(* IEC 61131-3 sources: Mizera_Tube/Plc (part 11) *)

(* ---- DataInterp.plc ---- *)
*******************************************************************************
*   DataInterp.plc
*   ESAutomotion
*   LASER machine
*******************************************************************************
#funcdec "DynMng.plc"

VAR
#include "Cnc.inc"

END_VAR

VAR_IN_OUT
#include "mem.inc"
END_VAR

#include "Iol.inc"

VAR_IN_OUT
A_CUT_DISTANCE          AT %L_CutDistance;
A_CUT_PRESSURE          AT %L_CutPressure;
A_CUT_FOCAL             AT %L_CutFocal;
A_CUT_FEED              AT %L_FeedA;
A_CUT_POWER             AT %L_CutPower;
A_CUT_DUTY              AT %L_CutDuty;
A_OPTION_FUN_SPEED      AT %L_SourceInt16;
A_OPTION_ENAB           AT %L_SourceInt16;
END_VAR

VAR
END_VAR

*******************************************************************************
*   Calcola dati di taglio tramite interpolazione lineare tra 2 linee di taglio
*
*       Formula: Y = Y1 + ( ((X-X1)/(X2-X1)) * (Y2-Y1) )
*******************************************************************************
FUNCTION_BLOCK LSR_DATA_INTERP

VAR_INPUT
xAngle:         DWORD;      * degree x 1000
xCutLineInd:    DWORD;      *
xFir:           DWORD;      *
END_VAR

VAR_OUTPUT
yCutPower:      DWORD;
yCutDuty:       DWORD;
yCutPressure:   DWORD;
yCutFocal:      DWORD;
yCutDistance:   DWORD;
yCutFeed:       DWORD;
yCutFeedPerc:   DWORD;
yFirstLine:     DWORD;
ySecondLine:    DWORD;
END_VAR

VAR
lAngleABS:      DWORD;
lFirstCutLine:  DWORD;
lSecondCutLine: DWORD;
l_x1:           DWORD;
l_x2:           DWORD;
l_y1:           DWORD;
l_y2:           DWORD;
l_x_x1:         DWORD;
l_x2_x1:        DWORD;
l_y2_y1:        DWORD;
POWER_CALC:     POINTS_INT_CALC;
POWER_CALC2:    POINTS_INT_CALC;
DUTY_CALC:      POINTS_INT_CALC;
DUTY_CALC2:     POINTS_INT_CALC;
Fir1:           DWORD;
flgerror_fir1:  DWORD;
RTRIG_FIR_INIT: R_TRIG;
l_CutFeedPerc:  DWORD;
ltemp:          DWORD;
END_VAR
***************************************

CAL  RTRIG_FIR_INIT (CLK:=%cn0.rc8.0)
LD   RTRIG_FIR_INIT.Q
JMPCN no_init_fir

LD   xFir
DIV  %plc0.PlcCycle
ST   Fir1
LD   0
FIR_INIT (INS=7, LEN=Fir1)
ST   flgerror_fir1             * 0 = OK

no_init_fir:
LD   xAngle
ABS
ST   lAngleABS

LD   lAngleABS
GE   30000
JMPCN no_30
LD   5
ST   lFirstCutLine
LD   6
ST   lSecondCutLine

LD   30000
ST   l_x1
LD   45000
ST   l_x2
JMP  com_a

no_30:
LD   lAngleABS
GE   15000
JMPCN no_15
LD   xCutLineInd
ST   lFirstCutLine
LD   5
ST   lSecondCutLine
LD   15000
ST   l_x1
LD   30000
ST   l_x2
JMP  com_a

no_15:
LD   xCutLineInd
ST   lFirstCutLine
ST   lSecondCutLine
LD   0
ST   l_x1
LD   15000
ST   l_x2

com_a:
LD   lAngleABS
SUB  l_x1
ST   l_x_x1
LD   l_x2
SUB  l_x1
ST   l_x2_x1

LD   lFirstCutLine
ST   yFirstLine
LD   lSecondCutLine
ST   ySecondLine

***************************************
*   Pressione
***************************************
PATH %TabLsr[lFirstCutLine]
LD   A_CUT_PRESSURE
ST   l_y1

PATH %TabLsr[lSecondCutLine]
LD   A_CUT_PRESSURE
ST   l_y2

LD   l_y2
SUB  l_y1
ST   l_y2_y1

LD   l_x_x1
MULDIV(M=l_y2_y1,D=l_x2_x1)
ADD  l_y1
ST   yCutPressure

***************************************
*   Focale
***************************************
PATH %TabLsr[lFirstCutLine]
LD   A_CUT_FOCAL
ST   l_y1

PATH %TabLsr[lSecondCutLine]
LD   A_CUT_FOCAL
ST   l_y2

LD   l_y2
SUB  l_y1
ST   l_y2_y1

LD   l_x_x1
MULDIV(M=l_y2_y1,D=l_x2_x1)
ADD  l_y1
ST   yCutFocal

***************************************
*   Altezza di taglio
***************************************
PATH %TabLsr[lFirstCutLine]
LD   A_CUT_DISTANCE
ST   l_y1

PATH %TabLsr[lSecondCutLine]
LD   A_CUT_DISTANCE
ST   l_y2

LD   l_y2
SUB  l_y1
ST   l_y2_y1

LD   l_x_x1
MULDIV(M=l_y2_y1,D=l_x2_x1)
ADD  l_y1
ST   yCutDistance

***************************************
*   Velocita' di taglio
*   - yCutFeed  [mm/min]
*   - yCutFeedPerc  [%] rispetto a linea taglio no bevel
***************************************
***todo PATH %TabLsr[lFirstCutLine]
PATH %TabLsr[1]
LD   A_CUT_FEED
ST   l_y1

PATH %TabLsr[lSecondCutLine]
LD   A_CUT_FEED
ST   l_y2

LD   l_y2
SUB  l_y1
ST   l_y2_y1

LD   lAngleABS
ST   l_x_x1
LD   l_x2
ST   l_x2_x1

LD   l_x_x1
MULDIV(M=l_y2_y1,D=l_x2_x1)
ADD  l_y1
ST   yCutFeed

LD   100            * 100%
ST   l_CutFeedPerc

LD   yCutFeed
MUL  100
DIV  l_y1
ST   l_CutFeedPerc

***todo
***LD   l_y2_y1
***EQ   0
***JMPC f_eq
***LD   yCutFeed
***SUB  l_y1
***MUL  100
***DIV  l_y2_y1

LD   0                       * N/C
FIR_RUN (INS=7, X=l_CutFeedPerc)
ST   ltemp

LD   l_CutFeedPerc
EQ   2147483647
JMPCN no_err_1

LD   ltemp
ST   l_CutFeedPerc

no_err_1:
f_eq:
LD   l_CutFeedPerc
ST   yCutFeedPerc

***************************************
*   Potenza
***************************************
PATH %TabLsr[lFirstCutLine]

LD   A_CUT_POWER
ST   l_y1

LD   A_OPTION_FUN_SPEED.3
JMPCN no_pow_funspeed

LD   PercInterpSpeed
ST   POWER_CALC.xPercSpeed
LD   lFirstCutLine
ST   POWER_CALC.xCutLineInd
LD   1
ST   POWER_CALC.xCodTec             * Tecnology 0=duty 1=power 2=frequency

CAL  POWER_CALC

LD   POWER_CALC.yResult
DIV  1000
MUL  A_CUT_POWER
DIV  100
ST   l_y1

no_pow_funspeed:

PATH %TabLsr[lSecondCutLine]
LD   A_CUT_POWER
ST   l_y2

LD   A_OPTION_FUN_SPEED.3           * enab power=funz(speed)
JMPCN no_pow_funspeed2

LD   PercInterpSpeed
ST   POWER_CALC2.xPercSpeed
LD   lSecondCutLine
ST   POWER_CALC2.xCutLineInd
LD   1
ST   POWER_CALC2.xCodTec            * 0=duty 1=power 2=frequency

CAL  POWER_CALC2

LD   POWER_CALC2.yResult
DIV  1000
MUL  A_CUT_POWER
DIV  100
ST   l_y2

no_pow_funspeed2:
LD   l_y2
SUB  l_y1
ST   l_y2_y1

LD   l_x_x1
MULDIV(M=l_y2_y1,D=l_x2_x1)
ADD  l_y1
ST   yCutPower

***************************************
*   Duty
***************************************
PATH %TabLsr[lFirstCutLine]

LD   A_CUT_DUTY
ST   l_y1

LD   A_OPTION_FUN_SPEED.2           * enab duty=funz(speed)
JMPCN no_duty_funspeed

LD   PercInterpSpeed
ST   DUTY_CALC.xPercSpeed
LD   lFirstCutLine
ST   DUTY_CALC.xCutLineInd
LD   0
ST   DUTY_CALC.xCodTec              * 0=duty 1=power 2=frequency

CAL  DUTY_CALC

LD   DUTY_CALC.yResult
DIV  1000
MUL  A_CUT_DUTY
DIV  100
ST   l_y1

no_duty_funspeed:
PATH %TabLsr[lSecondCutLine]
LD   A_CUT_DUTY
ST   l_y2

LD   A_OPTION_FUN_SPEED.2           * enab duty=funz(speed)
JMPCN no_duty_funspeed2

LD   PercInterpSpeed
ST   DUTY_CALC2.xPercSpeed
LD   lSecondCutLine
ST   DUTY_CALC2.xCutLineInd
LD   0
ST   DUTY_CALC2.xCodTec             * 0=duty 1=power 2=frequency

CAL  DUTY_CALC2

LD   DUTY_CALC2.yResult
DIV  1000
MUL  A_CUT_DUTY
DIV  100
ST   l_y2

no_duty_funspeed2:
LD   l_y2
SUB  l_y1
ST   l_y2_y1

LD   l_x_x1
MULDIV(M=l_y2_y1,D=l_x2_x1)
ADD  l_y1
ST   yCutDuty

END_FUNCTION_BLOCK

*******************************************************************************
*   Calcola dati di taglio in base all'angolo utilizzando le pd_spline
*   dedicate nell'attuale linea di taglio selezionata
*
*NB:
*pd_spline[150]     potenza linea 1    	(L_SourceInt16.8=abilitazione)
*pd_spline[151]		velocità linea 1	(L_SourceInt16.9=abilitazione)
*pd_spline[152]		altezza linea 1	    (L_SourceInt16.10=abilitazione)
*pd_spline[153]		focale linea 1	    (L_SourceInt16.11=abilitazione)
*pd_spline[154]		duty linea 1	    (L_SourceInt16.12=abilitazione)
*pd_spline[155]		gas linea 1		    (L_SourceInt16.13=abilitazione)
*pd_spline[156]		... linea 1         (L_SourceInt16.14=abilitazione)
*
* NB: Usa variabili globali SOLO per la simulazione (PER TEST USO INTERNO!)
* NB: %LSRPlcOp0.3 -> Enab function
*******************************************************************************
FUNCTION_BLOCK LSRDATACALC_ANGLE

VAR_INPUT
xAngle:         DWORD;      * degree x 1000
xCutLineInd:    DWORD;      * cutting line selected (1-10)
END_VAR

VAR_OUTPUT
yCutPower:      DWORD;      * % x 1000
yCutDuty:       DWORD;      * % x 1000
yCutFocal:      DWORD;      * % x 1000
yCutCuth:       DWORD;      * % x 1000
yCutGas:        DWORD;      * % x 1000
END_VAR

VAR
lAngleABS:      DWORD;
pdspline_num:   DWORD;
tmpPower:       DWORD;
tmpDuty:        DWORD;
tmpFocal:       DWORD;
tmpCuth:        DWORD;
tmpGas:         DWORD;
ANGLE_POWER_CALC:   LINEAR_CALC;
ANGLE_DUTY_CALC:    LINEAR_CALC;
ANGLE_FOCAL_CALC:   LINEAR_CALC;
ANGLE_CUTH_CALC:    LINEAR_CALC;
ANGLE_GAS_CALC:     LINEAR_CALC;
END_VAR
***************************************

*** SOLO per SIMULAZIONE INTERNA
LD   %TsCutDataLinear.CDL_SimOnPsw
EQ   2021
JMPCN no_sim_datainterp

LD   %TsCutDataLinear.CDL_SimAngle
ST   lAngleABS

LD   1
ST   xCutLineInd            * 1 per solo TEST !

JMP  initf

no_sim_datainterp:
LD   xAngle
ABS
ST   lAngleABS

initf:
PATH %TabLsr[xCutLineInd]

* Cuttting lines 1,2,3
LD   xCutLineInd
SUB  1
MUL  7                      * numero pd_spline[] per ciascuna linea di taglio
ADD  150
ST   pdspline_num           * 150 pd_spline linea1, 157 pd_spline linea2.....

* Cutting lines 11,12,13
LD   xCutLineInd
GT   10
JMPCN FROM11TO15
     LD   xCutLineInd
     SUB  11
     MUL  7                 * numero pd_spline[] per ciascuna linea di taglio
     ADD  180
     ST   pdspline_num      * 180 pd_spline linea1, 157 pd_spline linea2.....
FROM11TO15:

***************************************
*   POTENZA
*   pd_spline[150]=linea 1
*   Il valore trovato è l'incremento o
*   decremento della potenza attuale
***************************************
LD   0
ST   tmpPower

LD   A_OPTION_ENAB.8
AND  %LSRPlcOp0.3                       * Enab data cutting interpolation
AND  IncaseofbevelCut
JMPCN dato_ko

LD   lAngleABS
ST   ANGLE_POWER_CALC.xInput

LD   pdspline_num
ST   ANGLE_POWER_CALC.xIndex

CAL  ANGLE_POWER_CALC

LD   ANGLE_POWER_CALC.yResult
EQ   2147483647
JMPC dato_ko

LD   ANGLE_POWER_CALC.yResult
ST   tmpPower

dato_ko:
LD   tmpPower
ST   yCutPower

***************************************
*   DUTY
*   pd_spline[154]=linea 1
*   Il valore trovato è l'incremento o
*   decremento del duty attuale
***************************************
LD   0
ST   tmpDuty

LD   A_OPTION_ENAB.12
AND  %LSRPlcOp0.3                       * Enab data cutting interpolation
AND  IncaseofbevelCut
JMPCN dato_ko1

LD   lAngleABS
ST   ANGLE_DUTY_CALC.xInput

LD   pdspline_num
ADD  4
ST   ANGLE_DUTY_CALC.xIndex

CAL  ANGLE_DUTY_CALC

LD   ANGLE_DUTY_CALC.yResult
EQ   2147483647
JMPC dato_ko1

LD   ANGLE_DUTY_CALC.yResult
ST   tmpDuty

dato_ko1:
LD   tmpDuty
ST   yCutDuty

***************************************
*   FOCALE
*   pd_spline[153]=linea 1
*   Il valore trovato è l'incremento o
*   decremento del duty attuale
***************************************
LD   0
ST   tmpFocal

LD   A_OPTION_ENAB.11
AND  %LSRPlcOp0.3                       * Enab data cutting interpolation
AND  IncaseofbevelCut
JMPCN dato_ko2

LD   lAngleABS
ST   ANGLE_FOCAL_CALC.xInput

LD   pdspline_num
ADD  3
ST   ANGLE_FOCAL_CALC.xIndex

CAL  ANGLE_FOCAL_CALC

LD   ANGLE_FOCAL_CALC.yResult
EQ   2147483647
JMPC dato_ko2

LD   ANGLE_FOCAL_CALC.yResult
ST   tmpFocal

dato_ko2:
LD   tmpFocal
ST   yCutFocal

***************************************
*   ALTEZZA DI TAGLIO
*   pd_spline[152]=linea 1
*   Il valore trovato è l'incremento o
*   decremento del duty attuale
***************************************
LD   0
ST   tmpCuth

LD   A_OPTION_ENAB.10
AND  %LSRPlcOp0.3                       * Enab data cutting interpolation
AND  IncaseofbevelCut
JMPCN dato_ko3

LD   lAngleABS
ST   ANGLE_CUTH_CALC.xInput

LD   pdspline_num
ADD  2
ST   ANGLE_CUTH_CALC.xIndex

CAL  ANGLE_CUTH_CALC

LD   ANGLE_CUTH_CALC.yResult
EQ   2147483647
JMPC dato_ko3

LD   ANGLE_CUTH_CALC.yResult
ST   tmpCuth

dato_ko3:
LD   tmpCuth
ST   yCutCuth

***************************************
*   GAS
*   pd_spline[155]=linea 1
*   Il valore trovato è l'incremento o
*   decremento della pressione attuale
***************************************
LD   0
ST   tmpGas

LD   A_OPTION_ENAB.13
AND  %LSRPlcOp0.3                       * Enab data cutting interpolation
AND  IncaseofbevelCut
JMPCN dato_ko4

LD   lAngleABS
ST   ANGLE_GAS_CALC.xInput

LD   pdspline_num
ADD  5
ST   ANGLE_GAS_CALC.xIndex

CAL  ANGLE_GAS_CALC

LD   ANGLE_GAS_CALC.yResult
EQ   2147483647
JMPC dato_ko4

LD   ANGLE_GAS_CALC.yResult
ST   tmpGas

dato_ko4:
LD   tmpGas
ST   yCutGas

END_FUNCTION_BLOCK

*******************************************************************************
*   GESTIONE DI UNA FUNZIONE LINEARE GENERICA
*   DATO UN PUNTO (X o Y) VIENE CALCOLATO IL RELATIVO PUNTO (Y o X)
*
*   UTILIZZATA PER IL CALCOLO DI UNA CORREZIONE DI TEMPO SUL FILTRO FIR DI
*   SINCRONISMO TRA VELOCITA' E DUTY IN BASE ALL FREQUENZA IMPOSTATA.
*   Questo perchè normalmente il generatore, per il DUTY, ha un tempo di risposta
*   diverso in funzione della frequenza settata
*
*       LinearFun_tim_Y1        AT %rGui22;     *(rGui22)Funzione lineare: Y1
*       LinearFun_tim_Y2        AT %rGui23;     *(rGui23)Funzione lineare: Y1
*       LinearFun_freq_X1       AT %rGui24;     *(rGui24)Funzione lineare: X1
*       LinearFun_freq_X2       AT %rGui25;     *(rGui25)Funzione lineare: X4
*       LinearFun_freq_REF      AT %rGui26;     *(rGui26)Funzione lineare: frequenza di riferimento per settaggio tempo sync duty=fun(vel)
*
*       Formula: Y = Y1 + ( ((X-X1)/(X2-X1)) * (Y2-Y1) )
*
*******************************************************************************
FUNCTION_BLOCK LSR_GEN_LIN_INTERP

VAR_INPUT
x_Y1:           DWORD;
x_Y2:           DWORD;
x_X1:           DWORD;
x_X2:           DWORD;
x_X:            DWORD;
x_REF:          DWORD;
END_VAR

VAR_OUTPUT
y_Y:            DWORD;
y_REF:          DWORD;
END_VAR

VAR
l_xref_x1:      DWORD;
l_x_x1:         DWORD;
l_x2_x1:        DWORD;
l_y2_y1:        DWORD;
temp:           DWORD;
END_VAR
***************************************

LD   x_X
SUB  x_X1
ST   l_x_x1

LD   x_REF
SUB  x_X1
ST   l_xref_x1

LD   x_X2
SUB  x_X1
ST   l_x2_x1

LD   x_Y2
SUB  x_Y1
ST   l_y2_y1

LD   l_x_x1
MULDIV(M=l_y2_y1,D=l_x2_x1)
ST   temp

LD   temp
ADD  x_Y1
ST   y_Y

LD   l_xref_x1
MULDIV(M=l_y2_y1,D=l_x2_x1)
ST   temp

LD   temp
ADD  x_Y1
ST   y_REF

END_FUNCTION_BLOCK

(* ---- DynMng.plc ---- *)
*******************************************************************************
*   DynMng.plc
*   ESAutomotion
*   LASER machine
*******************************************************************************
VAR
#include "Cnc.inc"
END_VAR

VAR_IN_OUT
#include "mem.inc"
END_VAR

#include "Iol.inc"

VAR
END_VAR

*******************************************************************************
*
*******************************************************************************
FUNCTION_BLOCK PERC_CALC

VAR_INPUT
xAct:         DWORD;          * actual value
xSet:         DWORD;          * programmed value
END_VAR

VAR_OUTPUT
yPercSpeed:   DWORD;          * percentual value
END_VAR

VAR
END_VAR

LD   xAct                          ** actual value
MUL  200
ADD  1000
DIV  2
DIV  (
LD   xSet                          ** programmed value
MUL  1000
DIV  60                       * [mm/s]
)
MUL  1000
ST   yPercSpeed                    ** percentual value

END_FUNCTION_BLOCK

FUNCTION_BLOCK POINTS_INT_CALC

VAR_INPUT
xPercSpeed:   DWORD;          * Speed percentual value
xCutLineInd:  DWORD;          * cut line index (initial value 1 to 10)
xCodTec:      DWORD;          * Tecnology 0=duty 1=power 2=frequency
END_VAR

VAR_OUTPUT
yResult:      DWORD;          * Result
yOk:          DWORD;          * error code
END_VAR

VAR
Index:        DWORD;          * index of the technology table (xCutLineInd-1)*4 + xCodTec
InsNum:       DWORD;          * Istance number
PolResut:     DWORD;          * Polynomial result
Segment:      DWORD;          * Segment of the curve
segment_numb: DWORD;          * Segment number
END_VAR

LD   xCutLineInd                   ** cut line index (initial value 1 to 10)
SUB  1
MUL  4
ADD  xCodTec                       ** Tecnology 0=duty 1=power 2=frequency
ST   Index                         ** index of the technology table (xCutLineInd-1)*4 + xCodTec

LD   xCutLineInd
GT   11
JMPCN OUTOFTEN
     LD   Index
	 ADD  60
     ST   Index
OUTOFTEN:

LD   0
ST   Segment                       ** Segment of the curve

loop:

PATH %pd_splines[Index]            ** index of the technology table (xCutLineInd-1)*4 + xCodTec

LD   nSpan
SUB  1
ST   segment_numb                  ** Segment number

LD   Segment                       ** Segment of the curve
GT   segment_numb                  ** Segment number
OR  (
LD   Segment                       ** Segment of the curve
GT   20
)
JMPC check_last

PATH %pd_splines[Index]            ** index of the technology table (xCutLineInd-1)*4 + xCodTec
PATH %pd_spans[Segment]            ** Segment of the curve

LD   xPercSpeed                    ** Speed percentual value
LE   XSTART
JMPCN next_check

LD   YSTART                 * firts curve point
ST   yResult                       ** Result
JMP  exitfunc
next_check:

LD   xPercSpeed                    ** Speed percentual value
GT   XSTART
AND  (
LD   xPercSpeed                    ** Speed percentual value
LT   XEND
)
JMPC FindData

LD   xPercSpeed                    ** Speed percentual value
EQ   XSTART
JMPCN next_check1

LD   YEND
ST   yResult                       ** Result
JMP  exitfunc
next_check1:

LD   Segment                       ** Segment of the curve
ADD  1
ST   Segment                       ** Segment of the curve
JMP  loop

check_last:

LD   xPercSpeed                    ** Speed percentual value
GE   XEND
JMPCN gest_error
LD   YEND                 * firts curve point
ST   yResult                       ** Result
JMP  exitfunc

FindData:

LD   0
POLY_INIT (INS=1, XS=XSTART, XE=XEND, YS=YSTART, YE=YEND, A2=COEFICIENT_2, A3=COEFICIENT_3, A4=COEFICIENT_4, A5=COEFICIENT_5, PS=SPAN_NUM)
ST   PolResut                      ** Polynomial result

LD   PolResut                      ** Polynomial result
NE   0
JMPC gest_error

LD   0                      * N/C
POLY_EVAL_Y0 (INS=1, X0=xPercSpeed) ** Speed percentual value
ST   yResult                       ** Result

LD   yResult                       ** Result
EQ   2147483647
JMPCN exitfunc

gest_error:

LD  -1
ST  yOk                            ** error code
JMP exit
exitfunc:

LD   1
ST   yOk                           ** error code

exit:

END_FUNCTION_BLOCK

*******************************************************************************
* Generic linearization
*******************************************************************************
FUNCTION_BLOCK LINEAR_CALC

VAR_INPUT
xInput:         DWORD;          * Input value
xIndex:         DWORD;          * Spline index
END_VAR

VAR_OUTPUT
yResult:        DWORD;          * Result
yOk:            DWORD;          * error code
END_VAR

VAR
InsNum:         DWORD;          * Istance number
PolResut:       DWORD;          * Polynomial result
Segment:        DWORD;          * Segment of the curve
segment_numb:   DWORD;          * Segment number
END_VAR
*******************************************************************************
LD   0
ST   Segment                       ** Segment of the curve

LD   1
ST   yOk                           ** error code

LCloop:
PATH %pd_splines[xIndex]           ** Spline index

LD   nSpan
SUB  1
ST   segment_numb                  ** Segment number

LD   Segment                       ** Segment of the curve
GT   segment_numb                  ** Segment number
OR  (
LD   Segment                       ** Segment of the curve
GT   20
)
JMPC LCcheck_last

PATH %pd_splines[xIndex]           ** Spline index
PATH %pd_spans[Segment]            ** Segment of the curve

LD   xInput                        ** Input value
LE   XSTART
JMPCN LCnext_check

LD   YSTART                 * firts curve point
ST   yResult                       ** Result
JMP  LCexit

LCnext_check:
LD   xInput                        ** Input value
GT   XSTART
AND  (
LD   xInput                        ** Input value
LT   XEND
)
JMPC LCFindData

LD   xInput                        ** Input value
EQ   XSTART
JMPCN LCnext_check1

LD   YEND
ST   yResult                       ** Result
JMP  LCexit

LCnext_check1:
LD   Segment                       ** Segment of the curve
ADD  1
ST   Segment                       ** Segment of the curve
JMP  LCloop

LCcheck_last:
LD   xInput                        ** Input value
GE   XEND
JMPCN LCgest_error

LD   YEND                 * firts curve point
ST   yResult                       ** Result
JMP  LCexit

LCFindData:
LD   0
POLY_INIT(INS=5, XS=XSTART, XE=XEND, YS=YSTART, YE=YEND, A2=COEFICIENT_2, A3=COEFICIENT_3, A4=COEFICIENT_4, A5=COEFICIENT_5, PS=SPAN_NUM)
ST   PolResut                      ** Polynomial result

LD   PolResut                      ** Polynomial result
NE   0
JMPC LCgest_error

LD   0                      * N/C
POLY_EVAL_Y0(INS=5, X0=xInput)     ** Input value
ST   yResult                       ** Result

LD   yResult                       ** Result
EQ   2147483647
JMPCN LCexit

LCgest_error:
LD  -1
ST  yOk                            ** error code

LCexit:
END_FUNCTION_BLOCK

(* ---- FBAux.plc ---- *)
* CAL COMPARE(A:=,B:=)

FUNCTION_BLOCK     COMPARE

VAR_INPUT
A:                 DWORD;
B:                 DWORD;
END_VAR

VAR_OUTPUT
Q:                 BOOL;   * A>=B -> 1
yMax:              DWORD;
yMin:              DWORD;
END_VAR

LD   A
GE   B
ST   Q
JMPCN _CASE
     LD   A
     ST   yMax
	 LD   B
	 ST   yMin
JMP _COM
_CASE:
     LD   A
     ST   yMin
     LD   B
     ST   yMax
_COM:

END_FUNCTION_BLOCK

FUNCTION_BLOCK WARNING_ALM

VAR_INPUT
xVal: DWORD;
xWarnVal: DWORD;
xAlmVal: DWORD;
END_VAR

VAR_OUTPUT
yW: DWORD;
yA: DWORD;
END_VAR

VAR

END_VAR

LD  xAlmVal
GE  xWarnVal
JMPCN _LTNORMAL
    LD  xVal
	GT  xWarnVal
	ST  yW

	LD  xVal
	GT  xAlmVal
	ST  yA
_LTNORMAL:

LD  xAlmVal
LT  xWarnVal
JMPCN _GTNORMAL
    LD  xVal
	LT  xWarnVal
	ST  yW

	LD  xVal
	LT  xAlmVal
	ST  yA
_GTNORMAL:

*// Disable if inputs empty

LD  xAlmVal
AND xWarnVal
EQ  0
JMPCN _DISEN
    LD   0
    ST  yW
	ST  yA
_DISEN:

END_FUNCTION_BLOCK

* CAL FOC_SWLIM(xIn=,xMin=,xMax=)

FUNCTION_BLOCK FOC_SWLIM

VAR_INPUT
xIn: DWORD;
xMax: DWORD;
xMin: DWORD;
END_VAR

VAR_OUTPUT
Q: DWORD;
END_VAR

VAR
buffer: DWORD;
END_VAR

LD   xIn
ST   buffer

LD   xIn
GT   xMax
JMPCN _MAGGIORE
LD   xMax
ST   buffer
_MAGGIORE:

LD   xIn
LT   xMin
JMPCN _MINORE
LD   xMin
ST   buffer
_MINORE:

LD   buffer
ST   Q

END_FUNCTION_BLOCK

FUNCTION_BLOCK ANY_CLOCK_CHK

VAR_INPUT
xPeriod: DWORD;
xData: DWORD;
END_VAR

VAR_OUTPUT
Q: DWORD;
END_VAR

VAR
TON_CHK: TON;
buffer: DWORD;
buffer_1: DWORD;
Appoggio: BOOL;
END_VAR

LDN  TON_CHK.Q
ST   Appoggio
CAL  TON_CHK(IN:=Appoggio,PT:=xPeriod)
LD   TON_CHK.Q
JMPCN _LASTREC
     LD   xData
	 ST   buffer
_LASTREC:

LD   TON_CHK.ET
EQ (
LD   xPeriod
DIV  2
)
JMPCN _CURREC
     LD   xData
	 ST   buffer_1
_CURREC:

LD   buffer
EQ   buffer_1
ST   Q

END_FUNCTION_BLOCK

* CAL ABC_MINMAX(xA=,xB=,xC=)

FUNCTION_BLOCK ABC_MIN_MAX

VAR_INPUT
xA: DWORD;
xB: DWORD;
xC: DWORD;
END_VAR

VAR_OUTPUT
yMin: DWORD;
yMax: DWORD;
END_VAR

VAR
tem_A: DWORD;
tem_B: DWORD;
tem_C: DWORD;
buffer: DWORD;
END_VAR

LD   xA
ST   tem_A
LD   xB
ST   tem_B
LD   xC
ST   tem_C

LD   tem_A
GT   tem_B
JMPCN _SWAP_AB
     LD   tem_A
     ST   buffer

     LD   tem_B
     ST   tem_A

     LD   buffer
     ST   tem_B
_SWAP_AB:

LD   tem_A
GT   tem_C
JMPCN _SWAP_AC
     LD   tem_A
     ST   buffer

     LD   tem_C
     ST   tem_A

     LD   buffer
     ST   tem_C
_SWAP_AC:

LD   tem_B
GT   tem_C
JMPCN _SWAP_BC
     LD   tem_B
     ST   buffer

     LD   tem_C
     ST   tem_B

     LD   buffer
     ST   tem_C
_SWAP_BC:

LD   tem_A
ST   yMin

LD   tem_C
ST   yMax

END_FUNCTION_BLOCK

* CAL COSIN(In=,Angle=)

FUNCTION_BLOCK COSIN

VAR_INPUT
In: DWORD;
Angle: DWORD;
END_VAR

VAR_OUTPUT
Q: DWORD;
END_VAR

VAR
buffer: DWORD;
END_VAR

*LD   bevAngleHead1_calc1
LD   %C153
COS
ST   buffer

LD   In
MULDIV(M=1000,D=buffer)
ST   Q

END_FUNCTION_BLOCK

*//=============================================================================
*// CAL CALC_BLDFEED(xEn:=,xH:=,xV:=,xVPercent:=)
*//=============================================================================

FUNCTION_BLOCK CALC_BLD_FEED

VAR_INPUT
xEn:          BOOL;
xH:          DWORD;
xV:          DWORD;
xVPercent:   DWORD;
END_VAR

VAR
DIS_H:       DWORD;
DIS_V:       DWORD;
MinMax:    COMPARE;
END_VAR

VAR_OUTPUT
yPercent:    DWORD;
END_VAR

*//=============================================================================
*// Unloading Flaps On Each Support
*//=============================================================================
CAL  MinMax(A:=%gIso23,B:=%gIso24)

PATH %ax[xV]

LD   %ra24
SUB  %ax50.ra24
SUB  %ax61.ra24
ABS
ST   DIS_V

PATH %ax[xH]

LD   %ra24
SUB (
	 LD  MinMax.yMax
     MULDIV(M=1000,D=2)
)
ABS
ST   DIS_H

LD   100
ST   yPercent

LD   DIS_H
GT   DIS_V
AND  xEn
ANDN %ra3.0
ANDN %ra3.2
JMPCN _REDUCEV
     LD  DIS_V
	 MULDIV(M=100,D=DIS_H)
	 MULDIV(M=xVPercent,D=100)
     ST  yPercent      * 0-100%
_REDUCEV:

END_FUNCTION_BLOCK

(* ---- FBCutBox.plc ---- *)
#include "IolCutBox.inc"
#include "Iol.inc"

VAR
#include "RemContr.inc"
END_VAR

VAR_IN_OUT
#include "mem.inc"
BTN_START_CALIB         AT %Capacitive0.cButton0;    ** HMI
END_VAR

FUNCTION_BLOCK   PREC_CUTBOX

VAR_INPUT

xEcatNode:      DWORD;      * Ecat node where the cutbox is connected
xFocalPos:      DWORD;

xRefTravel:      BOOL;
xApplyNewFoc:    BOOL;
xPulReset:      BOOL;

END_VAR

VAR
FT_PRGRUN:              F_TRIG;
RTRIG_REQUEST:          R_TRIG;     ** HMI
RTRIG_CALIB:            R_TRIG;     ** Remote Controller

CalibRequest:           BOOL;   * Calib request
CALIBRAZIONE_RUN:       BOOL;   * Programma calibrazione in corso
END_VAR

VAR_OUTPUT
yExeCalib:              BOOL;   ** Calibration requested
yFarDistance:           BOOL;   ** Distance sensor outside the measurement range
yTipTouch:              BOOL;   ** Tip Touch error
END_VAR

CAL  FT_PRGRUN(CLK=PRGRUN_CN0)     ** M0.0 cn0.rc8.0  Programma in corso
CAL  RTRIG_REQUEST(CLK=BTN_START_CALIB) ** Calibration START button
CAL  RTRIG_CALIB(CLK:=RemContrCalib) ** Xhc_Puls.12 Execute calibration

LD   RTRIG_REQUEST.Q
OR   RTRIG_CALIB.Q                 ** Xhc_Puls.12 Execute calibration)
AND  MACC_TARATA                   ** (gPlc0.9)Assi tarati
OR   CalibRequest                  ** Calib request
S    CalibRequest                  ** Calib request

LD   M30_CN0                       ** M0.13 M30:EndProgram CN0
OR   MACC_ALARM                    ** (gPlc0.10)Macchina in allarme
OR   RESET_ALLARMI                 ** M100.4  Cancellazione allarmi attiva
OR   FT_PRGRUN.Q
R    CalibRequest                  ** Calib request

LD   CalibRequest                  ** Calib request
ST   CALIBRAZIONE_RUN              ** Programma calibrazione in corso
ST   yExeCalib                     ** Calibration requested

PATH  %ecat_ring0
PATH  %EcatNode[xEcatNode]

* FB Input Data

LD   xFocalPos
ST   PLC_FocalPosition

LD   xRefTravel
ST   DistanceReferenceTravel

LD   xApplyNewFoc
ST   FocusNewSetpoint

*

* // Cutbox to PLC ( INPUT )

LD   Ec_CutBoxST_ONE
ST   PLC_CutBoxST_ONE

LD   Ec_CutBoxST_TWO
ST   PLC_CutBoxST_TWO

LD   Ec_CutHeadST_ONE
ST   PLC_CutHeadST_ONE

LD   Ec_CutHeadST_TWO
ST   PLC_CutHeadST_TWO

LD   Ec_CutHeadSerST_ONE
ST   PLC_CutHeadSerST_ONE

LD   Ec_CutHeadSerST_TWO
ST   PLC_CutHeadSerST_TWO

* // ProCutter 2 settings

LD   Ec_ProCutterType
ST   PLC_ProCutterType

LD   Ec_StraylSensoProtWindGain
ST   PLC_StraylSensoProtWindGain

LD   Ec_ActualImageRatio
ST   PLC_ActualImageRatio

LD   Ec_CurrentFocalPosition.15   **YANG 241028 it is WORD
JMPC Focal_LT_ZERO
    LD   Ec_CurrentFocalPosition
    ST   PLC_CurrentFocalPosition
    JMP  Focal_GT_ZERO
Focal_LT_ZERO:
    LD  Ec_CurrentFocalPosition
    SUB  65536
    ST   PLC_CurrentFocalPosition
Focal_GT_ZERO:

LD   Ec_CustomerFocusOffset
ST   PLC_CustomerFocusOffset

*  // Distance functions

LD   Ec_WorkingDistance
ST   PLC_WorkingDistance

LD   Ec_NextCalibPosition
ST   PLC_NextCalibPosition

LD   Ec_PIDSpeedSetpoint
ST   PLC_PIDSpeedSetpoint

* // Sensor values

LD   Ec_TempProtectiveWindow
ST   PLC_TempProtWindow

LD   Ec_TemperatureFocusingLens
ST   PLC_TempFocusingLens

LD   Ec_TemperatureCollimatingLens
ST   PLC_TempCollimatingLens

LD   Ec_TemperatureCuttingHead
ST   PLC_TempCuttingHead

LD   Ec_TemperatureDistanceSensor
ST   PLC_TempDistanceSensor

LD   Ec_StraylightBeamPath
ST   PLC_StraylightBeamPath

LD   Ec_StraylightProtectWindowProc
ST   PLC_StraylProtectWindowProc

LD   Ec_StraylightProtectWindowCollima
ST   PLC_StrayLProtectWindowCol

LD   Ec_PresLeakProtectWindowProcess
ST   PLC_PresLeakProtectWindowProc

LD   Ec_ActualCuttingGasPres
ST   PLC_ActualCuttingGasPres

LD   Ec_HumidityInCuttingHead
ST   PLC_HumidityInCuttingHead

LD   Ec_Plasma
ST   PLC_Plasma

* Plc to Cutbox  (Output)

LD   xPulReset
R    DistanceCalibrateCharCurve

LD   DistanceCalibrateCharCurve
ST   Ec_CutBoxControl_ONE.0

LD   0
ST   Ec_CutBoxControl_ONE.1                 * SensorController

LD   NozzelLostCalibration                  * AT %CutBoxControl_ONE.3;
ST   Ec_CutBoxControl_ONE.3

LD   DistanceStrobeSignal                   * AT %CutBoxControl_ONE.4;
ST   Ec_CutBoxControl_ONE.4

LD   DistanceResetError                     *     AT %CutBoxControl_ONE.5;
ST   Ec_CutBoxControl_ONE.5

LD   ManualMode                            *    AT %CutBoxControl_ONE.6;
ST   Ec_CutBoxControl_ONE.6

LD   SyncToFieldbus                         *    AT %CutBoxControl_ONE.7;
ST   Ec_CutBoxControl_ONE.7

LD   CuttingHeadPower
ST   Ec_CutBoxControl_TWO.0

LD   SaveOutputData
ST   Ec_CutBoxControl_TWO.7

LD   DistanceReferenceTravel                 * AT %CuttHeadContr_ONE.0;
ST   Ec_CuttHeadContr_ONE.0

LD   FocusNewSetpoint
ST   Ec_CuttHeadContr_ONE.5                    * AT %CuttHeadContr_ONE.5;

LD   ResetPbus                             * AT %CuttHeadContr_ONE.7;
ST   Ec_CuttHeadContr_ONE.7

LD   ProcessDataSend
ST   PLC_CutHeadSerST_TWO.0

* ProCutter 2.0 control settings

LD   PLC_StraylightGainFactor
ST   Ec_StraylightGainFactor               *   AT %EcMDPOut7;

LD   PLC_MaxStrayLColLens
ST   Ec_MaxStraylightColLens               *   AT %EcMDPOut20;

LD   PLC_MaxStrayLProtWindowProc
ST   Ec_MaxStraylightProtWindowProcess      *   AT %EcMDPOut21;

LD   PLC_MaxHumidityCuttingHead
ST   Ec_MaxHumidityCuttingHead             *   AT %EcMDPOut22;

LD   PLC_MaxTempProtWindowProcess
ST   Ec_MaxTempProtWindowProcess           *   AT %EcMDPOut23;

LD   PLC_MaxTempCollimatingLens
ST   Ec_MaxTempCollimatingLens             *   AT %EcMDPOut24;

LD   PLC_MaxTempCuttingHead
ST   Ec_MaxTempCuttingHead                 *   AT %EcMDPOut26;

LD   PLC_MaxPresAssistGas
ST   Ec_MaxPressureAssistGas               *   AT %EcMDPOut27;

LD   PLC_MaxPresLeakProtWProc
ST   Ec_MaxPresLeakProtWProc               *   AT %EcMDPOut28;

LD   PLC_MaxStrayLCutHead
ST   Ec_MaxStrayLCutHead                   *    AT %EcMDPOut29;

LD   PLC_ImageRatio
ST   Ec_ImageRatio                        *    AT %EcMDPOut32;

LD   PLC_FocalPosition
ST   Ec_FocalPosition                     *    AT %EcMDPOut48;

* Distance function control settings

LD   PLC_SelectCharacteristicCurve     *   AT %SelectCharCurve;
ST   Ec_SelectCharacteristicCurve          *  AT %EcMDPOut6;

LD   PLC_DistanceFilterWindowSize      *   AT %DistFiltWindSize;
ST   Ec_DistanceFilterWindowSize           *  AT %EcMDPOut8;

LD   PLC_P_Parameter                  *   AT %P_Parameter;
ST   Ec_P_Parameter                       *  AT %EcMDPOut9;

LD   PLC_I_Parameter                  *   AT %I_Parameter;
ST   Ec_I_Parameter                       *  AT %EcMDPOut10;

LD   PLC_D_Parameter                  *   AT %D_Parameter;
ST   Ec_D_Parameter                       *  AT %EcMDPOut11;

LD   PLC_DistanceStandoffValue         *   AT %DistStandoffValue;
ST   Ec_DistanceStandoffValue              *  AT %EcMDPOut30;

LD   PLC_SpatterfilterTime            *    AT %SpatterfilterTime;
ST   Ec_SpatterfilterTime                 *  AT %EcMDPOut31;

LD   PLC_TipTouchLevel                *   AT %TipTouchLevel;
ST   Ec_TipTouchLevel                     *  AT %EcMDPOut33;

LD   PLC_MeasuringRangeLimit          *   AT %MeasRangeLimit;
ST   Ec_MeasuringRangeLimit               *  AT %EcMDPOut34;

LD   PLC_CollisionDelay               *   AT %CollisionDelay;
ST   Ec_CollisionDelay                    *  AT %EcMDPOut35;

LD   PLC_SetPointBand                 *   AT %SetPointBand;
ST   Ec_SetPointBand                      *  AT %EcMDPOut36;

LD   PLC_ControlDynamicBand           *    AT %ControlDynBand;
ST   Ec_ControlDynamicBand                *   AT %EcMDPOut37;

LD   PLC_MaxTemperatureSensorUnit      *    AT %MaxTempSensorUnit;
ST   Ec_MaxTemperatureSensorUnit           *  AT %EcMDPOut38;

LD  FarDistance
ST  yFarDistance                         ** Distance sensor outside the measurement range

LD   AlarmTipTouch
ST   yTipTouch

END_FUNCTION_BLOCK

(* ---- FBSpindl.plc ---- *)
*******************************************************************************
*   SpindFB.plc
*   ESAutomotion
*   LASER machine
*******************************************************************************
#funcdec "DynMng.plc"

VAR
#include "Cnc.inc"
END_VAR

VAR_IN_OUT
#include "mem.inc"
END_VAR

*******************************************************************************
*  FB chuck open close management
*  ---> The function block for pressure holding chuck
*******************************************************************************
FUNCTION_BLOCK SPINDLE

VAR_INPUT
xEmerg:             BOOL;
xProgRun:           BOOL;
xAutoClose:         BOOL;
xAutoOpen:          BOOL;
xManualClose:       BOOL;
xManualOpen:        BOOL;
xSpOpen:            BOOL;            * Sensor open
xSpClose:           BOOL;            * Sensor close
xCmdTime:           DWORD;           * Pressure holding time
xTimeout:           DWORD;

xThickness:         DWORD;
xResOut:            DWORD;
xIndGraphPress:     DWORD;
xFeedbkPress:       DWORD;
END_VAR

VAR_OUTPUT
yOpen:              BOOL;
yClose:             BOOL;            * NOT USED
yBrake:             BOOL;
yTimeout:           BOOL;
yPressAlm:          BOOL;

yAnOutPress:        DWORD;           * analog
yOutPressBar:       DWORD;           * [mbar]
yActualPressFeedbk: DWORD;           * [bar]
END_VAR

VAR
Appoggio:           BOOL;
req_open:           BOOL;
req_close:          BOOL;

InitOpen:           BOOL;
InitClosed:         BOOL;
Open:               BOOL;
Close:              BOOL;

R_TRIG_REQ_OP:      R_TRIG;
R_TRIG_REQ_CL:      R_TRIG;
R_TRIG_REQ_OP_AUT:  R_TRIG;
R_TRIG_REQ_CL_AUT:  R_TRIG;

TON_ALARM_TIMEOUT:  TON;
TON_ALARM_TIMEOUT1: TON;
TON_OPEN:           TON;
TON_CLOSE:          TON;

FindPress:    LINEAR_CALC;
END_VAR

* Init Condition

LD   ON_ONE_SCAN
AND  xSpOpen
S    InitOpen

LD   ON_ONE_SCAN
ANDN xSpOpen
S    InitClosed

*  Command

CAL  R_TRIG_REQ_OP (CLK:=xManualOpen)
CAL  R_TRIG_REQ_OP_AUT (CLK:=xAutoOpen)

LD   R_TRIG_REQ_OP.Q
OR   InitOpen
ANDN xProgRun
OR   xAutoOpen
*ANDN xEmerg
S    req_open

CAL  R_TRIG_REQ_CL (CLK:=xManualClose)
CAL  R_TRIG_REQ_CL_AUT (CLK:=xAutoClose)

LD   R_TRIG_REQ_CL.Q
OR   InitClosed
ANDN xProgRun
OR   xAutoClose
*ANDN xEmerg
R    req_open

**********************************************
* Output

LDN  xEmerg
ST   yBrake

LD   req_open
JMPCN no_open_req
     LD   ALWAYS_ONE
     S    Open
     R    Close
     R    InitOpen
     JMP  no_close_req
no_open_req:
     LD   ALWAYS_ONE
     S    Close
     R    InitClosed
     R    Open
no_close_req:

LD   Open
ANDN R_TRIG_REQ_OP.Q
ANDN R_TRIG_REQ_OP_AUT.Q
ST   yOpen
CAL  TON_ALARM_TIMEOUT (IN:=yOpen,PT:=xTimeout)

LD   Close
ANDN R_TRIG_REQ_CL.Q
ANDN R_TRIG_REQ_CL_AUT.Q
ST   yClose
CAL  TON_ALARM_TIMEOUT1 (IN:=yClose,PT:=xTimeout)

LD   TON_ALARM_TIMEOUT.Q
ANDN xSpOpen
OR(
LD   TON_ALARM_TIMEOUT1.Q
ANDN xSpClose
)
ST   yTimeout

* Close Pressure set

LD   xThickness
ST   FindPress.xInput

LD   xIndGraphPress
ST   FindPress.xIndex

CAL  FindPress

LD   FindPress.yResult
MUL  xResOut
DIV  10000          *10V
ST   yAnOutPress

LD   FindPress.yResult
ST   yOutPressBar   * [mbar]

************************************************************
* Pressure control

LD   xFeedbkPress
MUL  10000
DIV  4095
ST   yActualPressFeedbk

LD   FindPress.yResult
GT   (
LD   yActualPressFeedbk
ADD  500
)
OR  (
LD   FindPress.yResult
LT   (
LD   yActualPressFeedbk
SUB  500
)
)
ST   yPressAlm

END_FUNCTION_BLOCK

(* ---- FBSuppor.plc ---- *)
**********************************************
****** TUBE SUPPORTS MANAGEMENT **************
**********************************************

#include "usrMem.inc"
#include "Iol.inc"

VAR
#include "Cnc.inc"
END_VAR

VAR_IN_OUT
#include "usrIol.inc"
#include "mem.inc"
END_VAR

FUNCTION_BLOCK TUBE_SUPPORT

VAR_INPUT
xEmerg:	                     BOOL;
xAuto:	                     BOOL;
xUaxDir:                     BOOL;               * 1 - if spindle move towards the 0 of the machine decreasing its quota
                                                 * 0 - if spindle move towards the 0 of the machine increasing its quota
xSensorDwn:                  BOOL;               *Support is Down
xSensorOpen:	             BOOL;               *Support is Up
xManualUp: 	                 BOOL;               *Support Manual Up
xManualDwn:	                 BOOL;               *Support Manual Dwn
xManualOpen:                 BOOL;               *Clamps on Support Manual Open
xManualClose:                BOOL;               *Clamps on Support Manual Close
xAutoOpen:                   BOOL;               *Clamps on Support Auto Open
xAutoClose:                  BOOL;               *Clamps on Support Auto Close
xAutoUp:                     BOOL;               *Support Auto Up
xAutoDwn:                    BOOL;               *Support Auto Dwn
xAirPressure:                BOOL;               *For Both Support and Clamps Pressure Chk
xReset:                      BOOL;               *To Reset Allarm
xEnable:                     BOOL;

xPosU:	                     DWORD;              *U Axis Quota(ra4)
xSuperviseOft:               DWORD;              *Offset of position U to be closer to the support
xLimitQuota:	             DWORD;              *The Limit Forcing SupportS Dwn
xTimeOut:	                 DWORD;
END_VAR

VAR_OUTPUT
yAlarmDwn:                   BOOL;
yEvUp:	                     BOOL;
yEvDwn:	                     BOOL;
yHoldMovSuperv:              BOOL;
END_VAR

VAR
St_Up:	                     BOOL;
St_Down:	                 BOOL;
Ini_Down:	                 BOOL;
Ini_Up:                      BOOL;
AllowPosition:	             BOOL;

HoldSuperviAxis:            BOOL;
Supervise_Oft:              DWORD;

Ton_Down:                     TON;
RTRIG_ENAB:                R_TRIG;
END_VAR

* Added offset within safely down distance
LD   xSuperviseOft
ABS
ST   Supervise_Oft

LD   xSuperviseOft
ABS
GT   200000
JMPCN OUTRNGOFT
     LD   xSuperviseOft
	 ABS
     ST   Supervise_Oft
OUTRNGOFT:

LD   xUaxDir
JMPCN  no_check
     LD   xPosU
     SUB  200000                     * safety
     ADD  Supervise_Oft
     GT   xLimitQuota
     OR   ON_ONE_SCAN                ** PLCFLAGS.8  Flag on alla prima scansione PLC
     ST   AllowPosition

     LD   xPosU
     LT   xLimitQuota
     ANDN xSensorDwn
     ST   HoldSuperviAxis
no_check:

LDN  xUaxDir
JMPCN  no_check1
     LD   xPosU
     ADD  200000                     * safety
     SUB  Supervise_Oft
     LT   xLimitQuota
     OR   ON_ONE_SCAN                ** PLCFLAGS.8  Flag on alla prima scansione PLC
     ST   AllowPosition

     LD   xPosU
     GT   xLimitQuota
     ANDN xSensorDwn
     ST   HoldSuperviAxis
no_check1:

CAL  RTRIG_ENAB (CLK:=xEnable)
LD   ON_ONE_SCAN                     ** PLCFLAGS.8  Flag on alla prima scansione PLC
OR   RTRIG_ENAB.Q
AND  xSensorDwn
ST   Ini_Down

LD   ON_ONE_SCAN                     ** PLCFLAGS.8  Flag on alla prima scansione PLC
OR   RTRIG_ENAB.Q
ANDN xSensorDwn
ST   Ini_Up

***************************************
**** STATE VARIABLES ******************
***************************************

** UP STATE
LD  St_Down
AND(
LD  xAutoUp
OR(
LDN xAuto
AND xManualUp
)
)
AND xEmerg
OR(
LD   St_Up
ANDN St_Down
)
OR  Ini_Up
AND xEnable
ST  St_Up

** DWN STATE
LD  St_Up
AND(
LD  xAutoDwn
OR(
LDN xAuto
AND xManualDwn
)
)
ORN AllowPosition
AND xEmerg
OR(
LD   St_Down
ANDN St_Up
)
OR  Ini_Down
ST  St_Down

*******************************************

** OUTPUTS

LD  St_Up
AND AllowPosition
*AND xAirPressure
AND xEmerg
ST  yEvUp

LD  St_Down
ORN AllowPosition
*AND xAirPressure
AND xEmerg
ST  yEvDwn

** ALARMS

CAL Ton_Down(IN:=yEvDwn, PT=xTimeOut)
LD   Ton_Down.Q
ANDN xSensorDwn
S    yAlarmDwn

LD   xReset
OR   xSensorDwn
R    yAlarmDwn

** Hold the Supervisor

LD   HoldSuperviAxis
ST   yHoldMovSuperv

END_FUNCTION_BLOCK

(* ---- FBTimCnt.plc ---- *)
* Timer Function Block

FUNCTION_BLOCK TimCnt

VAR_INPUT
xEnable:          BOOL;  * To start the timer
xPreset:          BOOL;  * To preset the timer
xPreSec:         DWORD;  * Preset timer value in seconds
xPreDay:         DWORD;  * Preset timer value in days
xMode:           DWORD;  * 0 == timer count up, 1 == timer count down
END_VAR

VAR_OUTPUT
yOutSec:         DWORD;  * Outputs in seconds
yOutDay:         DWORD;  * Outputs in days
END_VAR

VAR
Cnt_sec:         DWORD;
Cnt_day:         DWORD;
R_TRIG_CNTRST:  R_TRIG;
R_TRIG_CNT:     R_TRIG;
END_VAR

* Body of FB

CAL  R_TRIG_CNT (CLK:=%PLCFLAGS.10)

LD   xMode
EQ   0
JMPCN CNTUPCASE
     LD   R_TRIG_CNT.Q
     AND  xEnable
     JMPCN no_inc
          LD   Cnt_sec
          ADD  1
          ST   Cnt_sec
     no_inc:

     LD   Cnt_sec
     EQ   86400
     JMPCN no_day_inc
          LD   0
          ST   Cnt_sec

          LD   Cnt_day
          ADD  1
          ST   Cnt_day
     no_day_inc:
CNTUPCASE:

LD   xMode
NE   0
JMPCN CNTDWNCASE
     LD   R_TRIG_CNT.Q
     AND  xEnable
     ANDN(
     LD   Cnt_sec
     EQ   0
     )
     JMPCN no_inc_1
          LD   Cnt_sec
          SUB  1
          ST   Cnt_sec
     no_inc_1:

     LD   Cnt_sec
     EQ   0
     ANDN(
     LD   Cnt_day
     EQ   0
     )
     JMPCN no_day_inc_1
          LD   86400
          ST   Cnt_sec

          LD   Cnt_day
          SUB  1
          ST   Cnt_day
     no_day_inc_1:

CNTDWNCASE:

* Preset the timer result
CAL  R_TRIG_CNTRST (CLK:=xPreset)
LD   R_TRIG_CNTRST.Q
JMPCN PRESETCASE
LD   xPreSec
ST   Cnt_sec

LD   xPreDay
ST   Cnt_day
PRESETCASE:

* Outputs

LD   Cnt_sec
ST   yOutSec

LD   Cnt_day
ST   yOutDay

END_FUNCTION_BLOCK

(* ---- FLP.plc ---- *)
FUNCTION_BLOCK FF * Gestione Flip Flop di un ingresso

VAR_INPUT
xPulsante:      BOOL;
xResetState:    BOOL;
END_VAR

VAR_OUTPUT
yComandOn:      BOOL;
END_VAR

VAR
StepDueExec_A:  BOOL;
PulsOn_A:       BOOL;
RETAIN Comando: BOOL;
END_VAR

**********************************************************
* ---
LD   xPulsante     * Ingresso pulsante
AND  Comando       * stato interno del passo passo
ANDN PulsOn_A      * Mem.Pulsante Premuto
ANDN xResetState   * Forzatura Reset stato del Filp Flop
ST   StepDueExec_A * mem.Secondo step eseguito

LD   StepDueExec_A * mem.Secondo step eseguito
OR   xResetState   * Forzatura Reset stato del Filp Flop
R    Comando       * stato interno del passo passo

LD   xPulsante     * Ingresso pulsante
ANDN PulsOn_A      * Mem.Pulsante Premuto
ANDN StepDueExec_A * mem.Secondo step eseguito
S    Comando       * stato interno del passo passo

LD   xPulsante     * Ingresso pulsante
ST   PulsOn_A      * Mem.Pulsante Premuto

LD   Comando       * stato interno del passo passo
ST   yComandOn     * Comando On

END_FUNCTION_BLOCK

(* ---- Foc_Prec.plc ---- *)
*******************************************************************************
*   FOC_PREC.PLC
*******************************************************************************
#funcdec "DynMng.plc"
#funcdec "FBAux.plc"
#include "foc_prec.inc"

VAR
#include "Cnc.inc"
ValoreFocale:             DWORD;
FocLinearCalc:      LINEAR_CALC;
END_VAR

******************************************************************************
*   FUNZIONE LINEARIZZAZIONE FOCALE
*   Torna la variabile locale "ValoreFocale"
******************************************************************************
FUNCTION FOC_LIN

LD   %LSRPlcOp1.3
JMPCN NoCapLin

LD   128                            * FOCAL LINEARIZATION's pd_spline
ST   FocLinearCalc.xIndex

LD   ValoreFocale
ST   FocLinearCalc.xInput

CAL  FocLinearCalc

LD   FocLinearCalc.yResult
EQ   2147483647
JMPC NoCapLin
     LD   FocLinearCalc.yResult
     ST   ValoreFocale
NoCapLin:

END_FUNCTION

******************************************************************************
******************************************************************************
*   PRECITEC
*   Main function block used to regulate the focal lens
******************************************************************************
******************************************************************************
FUNCTION_BLOCK FOC_PRECITEC

VAR_INPUT
xReset:                  BOOL;
xAnRes:                 DWORD;
xCutFoc:                DWORD;
xFocal_Type:            DWORD;
xVal_Focale_ACT:        DWORD;
END_VAR

VAR
TP_CHK:                    TP;
TON_CHK:                  TON;
TON_REF_OK:               TON;      * Ritardo per conclusione reference precitec ok
TON_REF_ERR:              TON;      * Ritardo da inizio reference per bypass /error
TON_AUTO_ERR:             TON;      * Ritardo per emissione allarme errore in automatico
TON_REF_TIMEOUT:          TON;      * Durata azzeramento testa precitec
TON_SHAKEHAND_TIMEOUT:    TON;
TOF_REF_HEAD:             TOF;

appoggio:                BOOL;      * Appoggio condizioni start temporizzatore
Aux_ValoreFocale:       DWORD;
ValMemoFocale:          DWORD;

FOCLIM1:            FOC_SWLIM;
FOCLIM2:            FOC_SWLIM;
FOCLIM3:            FOC_SWLIM;
FOCLIM4:            FOC_SWLIM;
FOCLIM5:            FOC_SWLIM;
FOCLIM6:            FOC_SWLIM;
END_VAR

VAR_OUTPUT
yPrec_Pos_Run:           BOOL;
yFocAn:                 DWORD;
yMsg:                   DWORD;
yError:                 DWORD;
END_VAR

******************************************************************************
* PRECITEC: Homming Management
******************************************************************************
CAL  TOF_REF_HEAD (IN:=%PLCFLAGS.8,PT:=4000)
LD   xReset
OR   ForceRefGui
OR   TOF_REF_HEAD.Q
AND  (
LD   I_I_PREC_ERROR
ORN  I_I_PREC_POSITION_REACHED
)
S    O_O_PREC_REFERENCE

LD   I_I_PREC_POSITION_REACHED
AND  O_O_PREC_REFERENCE
ST   appoggio
CAL  TON_REF_OK(IN=appoggio,PT=2000)

LD   I_I_PREC_ERROR
AND  O_O_PREC_REFERENCE
ST   appoggio
CAL  TON_REF_ERR(IN=appoggio,PT=3000)
CAL  TON_REF_TIMEOUT(IN=O_O_PREC_REFERENCE,PT=6000)

LD   TON_REF_OK.Q
OR   TON_REF_ERR.Q
OR   TON_REF_TIMEOUT.Q
R    O_O_PREC_REFERENCE

******************************************************************************
*   PRECITEC: Automatic Focal Management
*   - Within plc cycle focal command checking
******************************************************************************
LD   xVal_Focale_ACT
ST   Aux_ValoreFocale

LDN  %cn0.rc8.0
JMPC Prec_Focale
     LD   xCutFoc
     ST   Aux_ValoreFocale
Prec_Focale:

LDN  TON_CHK.Q
ST   appoggio
CAL  TON_CHK(IN=appoggio, PT=%plc0.PlcCycle)
LD   TON_CHK.Q
JMPCN _AN_CHK
     LD   Aux_ValoreFocale
     ST   ValMemoFocale
_AN_CHK:

LD   Aux_ValoreFocale
NE   ValMemoFocale
ST   appoggio
CAL  TP_CHK(IN=appoggio,PT=20)
LD   TP_CHK.Q
ANDN O_O_PREC_REFERENCE
ST   O_O_PREC_AUTOMATIC

******************************************************************************
*   PRECITEC: FOCAL lens regulation
******************************************************************************

***************************************
*   125mm
***************************************
LD   xFocal_Type
EQ   125
JMPCN NO_PREC1
	 CAL  FOCLIM1(xIn=Aux_ValoreFocale,xMin=-9000,xMax=6000)
     LD   FOCLIM1.Q
	 ST   ValoreFocale

     FOC_LIN

     LD   ValoreFocale
     MULDIV(M=-6266,D=10000)
     ADD  4060
     ST   CntrlVoltage
NO_PREC1:

***************************************
*   150mm
***************************************
LD   xFocal_Type
EQ   150
JMPCN NO_PREC2
	 CAL  FOCLIM2(xIn=Aux_ValoreFocale,xMin=-13000,xMax=9000)
     LD   FOCLIM2.Q
	 ST   ValoreFocale

     FOC_LIN

     LD   ValoreFocale
     MULDIV(M=-4272,D=10000)
     ADD  4145
     ST   CntrlVoltage
NO_PREC2:

***************************************
*   175mm
***************************************
LD   xFocal_Type
EQ   175
JMPCN NO_PREC3
	 CAL  FOCLIM3(xIn=Aux_ValoreFocale,xMin=-18000,xMax=12000)
     LD   FOCLIM3.Q
	 ST   ValoreFocale

     FOC_LIN

     LD    ValoreFocale
     MULDIV(M=-3133,D=10000)
     ADD   4060
     ST    CntrlVoltage
NO_PREC3:

***************************************
*   200mm
***************************************
LD   xFocal_Type
EQ   200
JMPCN NO_PREC4
	 CAL  FOCLIM4(xIn=Aux_ValoreFocale,xMin=-26000,xMax=18000)
     LD   FOCLIM4.Q
	 ST   ValoreFocale

     FOC_LIN

     LD    ValoreFocale
     MULDIV(M=-2130,D=10000)
     ADD   3990
     ST    CntrlVoltage
NO_PREC4:

***************************************
*  500mm
***************************************
LD   xFocal_Type
EQ   500
JMPCN NO_PREC6
	 CAL  FOCLIM6(xIn=Aux_ValoreFocale,xMin=-10210,xMax=12790)
     LD   FOCLIM6.Q
	 ST   ValoreFocale

     FOC_LIN

     LD   ValoreFocale
     MULDIV(M=-4000,D=10000)
     ADD  5440
     ST   CntrlVoltage
NO_PREC6:

* Cumulative focal value on output

LD   CntrlVoltage
MULDIV(M=xAnRes,D=10000)
ST   yFocAn

LDN  O_O_PREC_REFERENCE
ANDN I_I_PREC_POSITION_REACHED
ST   yPrec_Pos_Run
CAL  TON_SHAKEHAND_TIMEOUT(IN=yPrec_Pos_Run, PT=4000)

******************************************************************************
* Alarm and Messages
******************************************************************************
LD   TON_REF_ERR.Q
ST   yError.0

LD   TON_REF_TIMEOUT.Q
ST   yError.1

LD   I_I_PREC_ERROR
ST   yError.2

LDN  I_I_PREC_SW1
ORN  I_I_PREC_SW4
ST   yError.3

LD   TON_SHAKEHAND_TIMEOUT.Q
ST   yError.4

LDN  I_I_PREC_SW1
ST   yMsg.0

LDN  I_I_PREC_SW4
ST   yMsg.1

LD   TON_REF_OK.Q
ST   yMsg.2

******************************************************************************
*   PRECITEC: Updating user interface informations
******************************************************************************
LD   I_I_PREC_ERROR
ST   %fLeds.0

LD   I_I_PREC_POSITION_REACHED
ST   %fLeds.1

LD   O_O_PREC_REFERENCE
ST   %fLeds.2

LD   O_O_PREC_AUTOMATIC
ST   %fLeds.3

END_FUNCTION_BLOCK
******************************************************************************

(* ---- FocProco.plc ---- *)
*******************************************************************************
*   FOCPROCO.PLC
*   ESAutomotion
*   LASER machine
*******************************************************************************
#funcdec "DynMng.plc"

VAR
#include "Cnc.inc"

TempFocalValue: DWORD;                      * Temporary value focal

PwmLinearCalc:  LINEAR_CALC;

END_VAR

#include "Iol.inc"
#include "LsrGest.inc"

VAR_IN_OUT

#include "mem.inc"

Min             AT %pwPar0;         * Minimum value (x.xxx mm)
Max             AT %pwPar1;         * Maximum value (x.xxx mm)
DutyCalculated  AT %pwDutyCalcuSec; * Duty calculated (uSec)

Val_Focal_ACT   AT %TabLsr0.L_UserInt2;     * Last focal
END_VAR

*******************************************************************************
*   GESTIONE FOCALE con PWM
*******************************************************************************
FUNCTION_BLOCK FOC_PWM
VAR_INPUT
xId:            DWORD;              * 0,1
xSet:           DWORD;              * Focal setpoint (x.xxx mm)
xAct:           DWORD;              * Actual Focal value (x.xxx mm)
END_VAR

VAR_OUTPUT
yErr:           BOOL;       * Error
END_VAR

VAR
X2_X1Temp:      DWORD;
Y2_Y1Temp:      DWORD;
X_X1Temp:       DWORD;
END_VAR
*******************************************************************************

***PATH %FocalPwm[xId]

LD   xAct                          ** Actual Focal value (x.xxx mm)
GT   Max                           ** Maximum value (x.xxx mm)
OR (
LD   xSet                          ** Focal setpoint (x.xxx mm)
LT   Min                           ** Minimum value (x.xxx mm)
)
JMPCN NoOutOf

LD   0                  * Default = 0
ST   xAct                          ** Actual Focal value (x.xxx mm)

NoOutOf:
LD   xSet                          ** Focal setpoint (x.xxx mm)
GT   Max                           ** Maximum value (x.xxx mm)
OR (
LD   xSet                          ** Focal setpoint (x.xxx mm)
LT   Min                           ** Minimum value (x.xxx mm)
)
ST   yErr                          ** Error

LD   yErr                          ** Error
JMPCN NoOutOf2

LD   xAct                          ** Actual Focal value (x.xxx mm)
ST   xSet                          ** Focal setpoint (x.xxx mm)

NoOutOf2:
LD   838                * Set 50Hz
ST   HW2_FREQ

LD   16#0fff            * 12 bit of resolution
ST   HW2_PWM_RES

LD   ALWAYS_ONE                    ** PLCFLAGS.1  Flag sempre stato on
ST   HW2_PWM_CFG_EN

***************************************
*   PWM calc
***************************************
LD   xSet                          ** Focal setpoint (x.xxx mm)
ST   PwmLinearCalc.xInput

LD   139                            * pd_spline
ST   PwmLinearCalc.xIndex

CAL  PwmLinearCalc

LD   PwmLinearCalc.yResult
EQ   2147483647
JMPCN DatoOk

LD   0
ST   DutyCalculated                ** Duty calculated (uSec)
JMP  NoLin

DatoOk:
LD   PwmLinearCalc.yResult
DIV  1000
ST   DutyCalculated                ** Duty calculated (uSec)

NoLin:
LD   DutyCalculated                ** Duty calculated (uSec)
MUL  10000
DIV  48828           * 1 point = 4,8828125uSec
AND  16#0fff
ST   HW2_PWM_DUTY

END_FUNCTION_BLOCK

***
VAR
FOC_PWM_0:   FOC_PWM;                    * focal FB
END_VAR

*******************************************************************************
*   GESTIONE FOCALE PROCON
*******************************************************************************
FUNCTION PROCON_FOCAL

LD   Val_Focal_ACT                 ** Last focal
ST   TempFocalValue                ** Temporary value focal

LD   MACCH_IN_MANUALE              ** M100.24 SELEZIONE MACCHINA IN MANUALE
JMPC man_management

LD   %TabLsr0.L_CutFocal         ** Valore focale passato da tabelle
ST   TempFocalValue                ** Temporary value focal

man_management:

PATH %FocalPwm[0]

LD   TempFocalValue                ** Temporary value focal
ST   FOC_PWM_0.xSet

CAL  FOC_PWM_0                     ** focal FB

LD   FOC_PWM_0.yErr
S    %PLCerr5.31

LD   RESET_ALLARMI                 ** M100.4  Cancellazione allarmi attiva
R    %PLCerr5.31

END_FUNCTION

(* ---- intgraph.plc ---- *)
*******************************************************************************
*   INTGRAPH.PLC
*   ESAutomotion
*   LASER machine
*******************************************************************************
#funcdec "DynMng.plc"

VAR
#include "Cnc.inc"

Bevel0Calc:     LINEAR_CALC;
Bevel15Calc:    LINEAR_CALC;
Bevel30Calc:    LINEAR_CALC;
Bevel45Calc:    LINEAR_CALC;
PolResult:      DWORD;          * Polynomial result
Segment:        DWORD;          * Segment of the curve
segment_numb:   DWORD;          * Segment number
yResult:        DWORD;          * Result
yOk:            DWORD;          * error code
FTRIG_PGRRUN:   F_TRIG;
RTRIG_INIT:     R_TRIG;
END_VAR

VAR_IN_OUT
#include "mem.inc"
END_VAR

#include "Iol.inc"

*******************************************************************************
*   Gestione Sensore Capacitivo per linearizzazione da CNC (con bevel)
*   NOTA BENE: utilizza dati della struttura %TsCalib[]
*******************************************************************************
FUNCTION_BLOCK InterpGraph

VAR_INPUT
xInput:                  DWORD;
xActualAngle:            DWORD;
xIndexFirstTable:        DWORD;
xIndexSecondTable:       DWORD;
xIndexThirdTable:        DWORD;
xIndexFourthTable:       DWORD;
xIndexOutIntVal:         DWORD;
END_VAR

VAR_OUTPUT
yOutInterpVal:           DWORD;
END_VAR

PATH %pd_splines[xIndexOutIntVal]

LD   3
ST   nSpan

LD   0
ST   Segment                       ** Segment of the curve

loop1:

PATH %pd_splines[xIndexOutIntVal]
PATH %pd_spans[Segment]            ** Segment of the curve

LD   1
ST   SPAN_NUM

LD   0
ST   COEFICIENT_0
ST   COEFICIENT_1
ST   COEFICIENT_2
ST   COEFICIENT_3
ST   COEFICIENT_4
ST   COEFICIENT_5

LD   Segment                       ** Segment of the curve
ADD  1
ST   Segment                       ** Segment of the curve

LD   Segment                       ** Segment of the curve
LT   4
JMPC loop1

***************************************
*   0 degree
***************************************
LD   xInput
MUL  1000
ST   Bevel0Calc.xInput

LD   xIndexFirstTable
ST   Bevel0Calc.xIndex

CAL  Bevel0Calc

PATH %pd_splines[xIndexOutIntVal]
PATH %pd_spans0

LD   0
ST   XSTART
LD   %TsCalib1.targ_b_axis              * es. 15 gradi
ST   XEND

LD   Bevel0Calc.yResult                * Result
ST   YSTART

***************************************
*   15 degree
***************************************
LD   xInput
MUL  1000
ST   Bevel15Calc.xInput

LD   xIndexSecondTable
ST   Bevel15Calc.xIndex

CAL  Bevel15Calc

PATH %pd_splines[xIndexOutIntVal]
PATH %pd_spans0

LD   Bevel15Calc.yResult                * Result
ST   YEND

PATH %pd_splines[xIndexOutIntVal]
PATH %pd_spans1

LD   %TsCalib1.targ_b_axis              * es. 15 gradi
ST   XSTART
LD   %TsCalib2.targ_b_axis              * es. 30 gradi
ST   XEND

LD   Bevel15Calc.yResult                * Result
ST   YSTART                     * Height 15 degree bevel

***************************************
*   30 degree
***************************************
LD   xInput
MUL  1000
ST   Bevel30Calc.xInput

LD   xIndexThirdTable
ST   Bevel30Calc.xIndex

CAL  Bevel30Calc

PATH %pd_splines[xIndexOutIntVal]
PATH %pd_spans1

LD   Bevel30Calc.yResult               * Result
ST   YEND

PATH %pd_splines[xIndexOutIntVal]
PATH %pd_spans2

LD   %TsCalib2.targ_b_axis              * es. 30 gradi
ST   XSTART
LD   %TsCalib3.targ_b_axis              * es. 45 gradi
ST   XEND

LD   Bevel30Calc.yResult               * Result
ST   YSTART                    * Height 30 degree bevel

***************************************
*   45 degree
***************************************
LD   xInput
MUL  1000
ST   Bevel45Calc.xInput

LD   xIndexFourthTable
ST   Bevel45Calc.xIndex

CAL  Bevel45Calc

PATH %pd_splines[xIndexOutIntVal]
PATH %pd_spans2

LD   Bevel45Calc.yResult               * Result
ST   YEND

PATH %pd_splines[xIndexOutIntVal]
PATH %pd_spans3

LD   Bevel45Calc.yResult               * Result
ST   YSTART                    * Height 45 degree bevel

LD   %TsCalib3.targ_b_axis              * es. 45 gradi
ST   XSTART

***************************************
LD   0
ST   Segment                       ** Segment of the curve

loop:

PATH %pd_splines[xIndexOutIntVal]

LD   nSpan
SUB  1
ST   segment_numb                  ** Segment number

LD   Segment                       ** Segment of the curve
GT   segment_numb                  ** Segment number
OR  (
LD   Segment                       ** Segment of the curve
GT   20
)
JMPC check_last

PATH %pd_splines[xIndexOutIntVal]
PATH %pd_spans[Segment]            ** Segment of the curve

LD   xActualAngle
LE   XSTART
JMPCN next_check

LD   YSTART                 * firts curve point
ST   yResult                       ** Result
JMP  exitfunc
next_check:

LD   xActualAngle
GT   XSTART
AND  (
LD   xActualAngle
LT   XEND
)
JMPC FindData

LD   xActualAngle
EQ   XSTART
JMPCN next_check1

LD   YEND
ST   yResult                       ** Result
JMP  exitfunc
next_check1:

LD   Segment                       ** Segment of the curve
ADD  1
ST   Segment                       ** Segment of the curve
JMP  loop

check_last:

LD   xActualAngle
GE   XEND
JMPCN gest_error
LD   YEND                   * firts curve point
ST   yResult                       ** Result
JMP  exitfunc

FindData:

LD   0
POLY_INIT (INS=2, XS=XSTART, XE=XEND, YS=YSTART, YE=YEND, A2=COEFICIENT_2, A3=COEFICIENT_3, A4=COEFICIENT_4, A5=COEFICIENT_5, PS=SPAN_NUM)
ST   PolResult                     ** Polynomial result

LD   PolResult                     ** Polynomial result
NE   0
JMPC gest_error

LD   0                      * N/C
POLY_EVAL_Y0 (INS=2, X0=xActualAngle)
ST   yResult                       ** Result

LD   yResult                       ** Result
EQ   2147483647
JMPCN exitfunc

gest_error:
LD  -1
ST  yOk                            ** error code
JMP exit
exitfunc:

LD   1
ST   yOk                           ** error code

exit:

LD   yResult                       ** Result
MUL  AnalCapFeedback       *Capacitive analog resolution
DIV  %LSRCostK31                   ** Capacitive sensor range
ST   yOutInterpVal

* Range for graph

LD   %LSRCostK31                   ** Capacitive sensor range
DIV  1000
ST   CapRange                      ** (C151) Capacitive range

* Reset interface command for coefficients calc

CAL  FTRIG_PGRRUN (CLK:=%cn0.rc8.0)

LD   FTRIG_PGRRUN.Q
JMPCN no_res_bit

LD   ALWAYS_ZERO                   ** PLCFLAGS.0  Flag sempre stato off
ST   CoefInterfCalc                ** (ui0.10) calculate the coefficients
no_res_bit:

END_FUNCTION_BLOCK

(* ---- IO_test.plc ---- *)
*******************************************************************************
*   IO_TEST.PLC
*   ESAutomotion
*   LASER machine
*******************************************************************************
VAR
#include "Cnc.inc"

*** Reserved from %C80 to %C99  !!!
*** Reserved from %R90 to %R99  !!!

MASK_IN0                AT %C80;        * C80 Forced Inputs
MASK_IN1                AT %C81;        * C81 Forced Inputs
MASK_IN2                AT %C82;        * C82 Forced Inputs
MASK_IN3                AT %C83;        * C83 Forced Inputs
MASK_IN4                AT %C84;        * C84 Forced Inputs
MASK_IN5                AT %C85;        * C85 Forced Inputs
MASK_IN6                AT %C86;        * C86 Forced Inputs
MASK_IN7                AT %C87;        * C87 Forced Inputs
MASK_IN8                AT %C88;        * C88 Forced Inputs
MASK_IN9                AT %C89;        * C89 Forced Inputs

MASK_OUT0               AT %C90;        * C90 Forced Outputs OFF/ON
MASK_OUT1               AT %C91;        * C91 Forced Outputs OFF/ON
MASK_OUT2               AT %C92;        * C92 Forced Outputs OFF/ON
MASK_OUT3               AT %C93;        * C93 Forced Outputs OFF/ON
MASK_OUT4               AT %C94;        * C94 Forced Outputs OFF/ON
MASK_OUT5               AT %C95;        * C95 Forced Outputs OFF/ON
MASK_OUT6               AT %C96;        * C96 Forced Outputs OFF/ON
MASK_OUT7               AT %C97;        * C97 Forced Outputs OFF/ON
MASK_OUT8               AT %C98;        * C98 Forced Outputs OFF/ON
MASK_OUT9               AT %C99;        * C99 Forced Outputs OFF/ON

ABIL_OUT0               AT %R90;        * R90 Enable single bit
ABIL_OUT1               AT %R91;        * R91 Enable single bit
ABIL_OUT2               AT %R92;        * R92 Enable single bit
ABIL_OUT3               AT %R93;        * R93 Enable single bit
ABIL_OUT4               AT %R94;        * R94 Enable single bit
ABIL_OUT5               AT %R95;        * R95 Enable single bit
ABIL_OUT6               AT %R96;        * R96 Enable single bit
ABIL_OUT7               AT %R97;        * R97 Enable single bit
ABIL_OUT8               AT %R98;        * R98 Enable single bit
ABIL_OUT9               AT %R99;        * R99 Enable single bit

ForceInputs             AT %C100.0;     * C100.0 Auxiliary to Force Inputs
ForceOutputs            AT %C100.1;     * C100.1 Auxiliary to Force Outputs

END_VAR

#include "Iol.inc"

VAR_IN_OUT
R_REGISTER              AT %R;          * R regsiter used about forcing output
C_REGISTER              AT %C;          * R regsiter used about forcing output
END_VAR

******************************************************************************
* INPUTS
******************************************************************************
FUNCTION_BLOCK INP_MNGMT
VAR_INPUT
xInp:       WORD;           *
xIndex:     WORD;           *
END_VAR

VAR_OUTPUT
yInp:       WORD;           *
END_VAR

VAR
IndexMask:  WORD;           *
END_VAR

LD   xIndex                        **
ADD  80
ST   IndexMask                     **

LD   C_REGISTER[IndexMask]         ** R regsiter used about forcing output
***Commentare OR se si vuole forzare a zero un ingresso
***OR   xInp
ST   yInp                          **

END_FUNCTION_BLOCK

******************************************************************************
* OUTPUTS
******************************************************************************
FUNCTION_BLOCK OUT_MNGMT
VAR_INPUT
xOut:       WORD;           *
xIndex:     WORD;           *
END_VAR

VAR_OUTPUT
yOut:       WORD;           *
END_VAR

VAR
IndexMask:  WORD;           *
SetResMask: WORD;           *
CncMask:    WORD;           *
END_VAR

LD   xIndex                        **
ADD  90
ST   IndexMask                     **

LD   ForceOutputs                  ** C100.1 Auxiliary to Force Outputs
JMPC EndOut

LD   0
ST   R_REGISTER[IndexMask]         ** R regsiter used about forcing output
ST   C_REGISTER[IndexMask]         ** R regsiter used about forcing output

EndOut:
LD   R_REGISTER[IndexMask]         ** R regsiter used about forcing output
AND  C_REGISTER[IndexMask]         ** R regsiter used about forcing output
ST   SetResMask                    **

LD   R_REGISTER[IndexMask]         ** R regsiter used about forcing output
XOR  16#FFFF                       ** bit complement
AND  xOut                          **
ST   CncMask                       **

LD   SetResMask                    **
OR   CncMask                       **
ST   yOut                          **

END_FUNCTION_BLOCK

VAR
INP1:       INP_MNGMT;
INP2:       INP_MNGMT;
INP3:       INP_MNGMT;
INP4:       INP_MNGMT;
INP5:       INP_MNGMT;
INP6:       INP_MNGMT;
OUT1:       OUT_MNGMT;
OUT2:       OUT_MNGMT;
OUT3:       OUT_MNGMT;
OUT4:       OUT_MNGMT;
OUT5:       OUT_MNGMT;
END_VAR

******************************************************************************
FUNCTION INP_TEST
******************************************************************************
LD   ForceInputs                   ** C100.0 Auxiliary to Force Inputs
JMPCN BypassInp1

LD   %IW0
ST   INP1.xInp
LD   0
ST   INP1.xIndex
CAL  INP1
LD   INP1.yInp
ST   %IO0

LD   %IW1
ST   INP2.xInp
LD   1
ST   INP2.xIndex
CAL  INP2
LD   INP2.yInp
ST   %IO1

LD   %IW4
ST   INP3.xInp
LD   2
ST   INP3.xIndex
CAL  INP3
LD   INP3.yInp
ST   %IO4

LD   %IW5
ST   INP4.xInp
LD   3
ST   INP4.xIndex
CAL  INP4
LD   INP4.yInp
ST   %IO5

BypassInp1:
END_FUNCTION

******************************************************************************
FUNCTION OUT_TEST
******************************************************************************

LD   %QW2
ST   OUT1.xOut
LD   0
ST   OUT1.xIndex
CAL  OUT1
LD   OUT1.yOut
ST   %QW2

LD   %QW3
ST   OUT2.xOut
LD   1
ST   OUT2.xIndex
CAL  OUT2
LD   OUT2.yOut
ST   %IO3

LD   %QW6
ST   OUT3.xOut
LD   2
ST   OUT3.xIndex
CAL  OUT3
LD   OUT3.yOut
ST   %QW6

LD   %QW7
ST   OUT4.xOut
LD   3
ST   OUT4.xIndex
CAL  OUT4
LD   OUT4.yOut
ST   %QW7

END_FUNCTION

(* ---- LsrGest.plc ---- *)
*******************************************************************************
*   LSRGEST.PLC
*   ESAutomotion
*   LASER machine
*******************************************************************************
#funcdec "assi.plc"
#funcdec "canfb.plc"
#funcdec "cnc.plc"
#funcdec "mand.plc"
#funcdec "manrev.plc"
#funcdec "DynMng.plc"

VAR
#include "assi.inc"
#include "cnc.inc"
#include "RemContr.inc"

DutyCalc:   POINTS_INT_CALC;
PowerCalc:  POINTS_INT_CALC;
FreqCalc:   POINTS_INT_CALC;
PowerLin:   LINEAR_CALC;
END_VAR

VAR_IN_OUT
#include "mem.inc"
L_SOURCE16  AT %L_SourceInt16;
END_VAR

#include "iol.inc"
#include "LsrGest.inc"

*******************************************************************************
*   INTERPOLATION SPEED
*******************************************************************************
FUNCTION_BLOCK CALC_INTERP_SPEED
VAR_INPUT
xNumFir:            DWORD;		* 0,1,2 (numero fir=5+xNumFir)
xFir:               DWORD;
END_VAR

VAR_OUTPUT
yInterpSpeed:       DWORD;
END_VAR

VAR
interpSpeed:        DWORD;      * interpolation speed
firScan:            DWORD;      *
delScan:            DWORD;
RTRIG_FIR_INIT:     R_TRIG;
error:              DWORD;
nFir:               DWORD;
END_VAR

LD   %ax21.ra28                    * interpolator speed (micro/sec) Proc.Principale CN0
ST   interpSpeed                   ** interpolation speed

LD   5
ADD  xNumFir
ST   nFir

LD   %UnitWork.gTravE
EQ   1
JMPCN no_pipe1
LD   %ax21.ra30                    * tcp speed (micro/sec)
ST   interpSpeed                   ** interpolation speed

no_pipe1:
* Filter on interpolated speed
LD   xFir
DIV  %plc0.PlcCycle         * plc scan
ST   firScan                       **

CAL  RTRIG_FIR_INIT (CLK:=%cn0.rc8.0)

LD   RTRIG_FIR_INIT.Q     * first scan
JMPCN no_init

LD   0               * N/C
FIR_INIT (INS=nFir, LEN=firScan)      **
ST   error             * 0 = OK

LD   %CostK26
DIV  %plc0.PlcCycle         * plc scan
ST   delScan                      **

LD   0
DELAY_INIT (INS=nFir, LEN=delScan)
ST   error

LD   error
NE   0
JMPC error_1

no_init:
LD   0                       * N/C
FIR_RUN (INS=nFir, X=interpSpeed)     ** interpolation speed
ST   yInterpSpeed

LD   yInterpSpeed
EQ   2147483647
JMPCN calc_

error_1:
LD   0
ST   yInterpSpeed

calc_:

LD   0
DELAY_RUN (INS=nFir,X=yInterpSpeed)
****DIV  10
ST  yInterpSpeed

END_FUNCTION_BLOCK

*******************************************************************************
*   LASER MANAGEMENT
*******************************************************************************
FUNCTION_BLOCK LSRGST

VAR_INPUT
xId:        DWORD;          * 0,1
xPower:     DWORD;          * Power
xDuty:      DWORD;          * Duty
xFreq:      DWORD;          * Frequency
END_VAR

VAR_OUTPUT
yEmission:  BOOL;           * Emission
END_VAR

VAR
corr_funz_speed:    BOOL;
appoggio:           BOOL;
tmpDutyLaserOut:    DWORD;      * Duty temp
tmpDutyLaserCmd:    DWORD;      * Duty temp commanded
tmpFreqLaserOut:    DWORD;      * Freq temp
tmpPowerLaserOut:   DWORD;      * Power temp
tmpPowerLaserCmd:   DWORD;      * Power temp commanded
appoggio_pow:       DWORD;
appoggio_duty:      DWORD;

RTRIG_EnVal1:       TRIG;
TRIG_EnVal1_G834:  TRIG;
TRIG_EnVal2_G834:  TRIG;
outputEnableON:     BOOL;       * Actually enable output (/pgm interrupted, etc..)
flyCutOnInitPulse:  BOOL;
R_TRIG_FC_ON_INIT:  R_TRIG;
shoot_fly_on:       BOOL;       * to disable shoot in hold during fly cut old board
TOF_Pul_Stop:       TOF;

Strobe_Funz_M410:   BOOL;
Strobe_Funz_M411:   BOOL;
R_TRIG410:          R_TRIG;     * Emission ON Laser
R_TRIG411:          R_TRIG;     * Emission OFF Laser
FTRIG_STOP:         F_TRIG;

END_VAR
*******************************************************************************

PATH %TabLsr[CurrentLineExecute]

*******************************************************************************
*   M410 or TstP15.3 -> Emission ON
*******************************************************************************
LD   %cn0.rc9           ** Channel 0 M-Functions register
EQ   410
AND  %cn0.rc8.4         ** Channel 0 M-Functions Strobe
OR   LaserOn_REQ                   ** (TstP15.3) (LASER_ON)
ST   Strobe_Funz_M410

LD   %cn0.rc9           ** Channel 0 M-Functions register
EQ   411
AND  %cn0.rc8.4         ** Channel 0 M-Functions Strobe
OR   LaserOFF_REQ                  ** (TstP15.2) (LASER_OFF) Turn off laser from Iso
ST   Strobe_Funz_M411

CAL  R_TRIG410(CLK=Strobe_Funz_M410) ** Emission ON Laser
CAL  R_TRIG411(CLK=Strobe_Funz_M411) ** Emission OFF Laser

LD   R_TRIG410.Q    ** Fronte di salita M410 Attivazione Emission ON Laser
S    yEmission                     ** Emission

LD   R_TRIG411.Q    ** Fronte di salita M411 Disattivazione Emission ON Laser
ORN  PRGRUN_CN0                    ** M0.0 cn0.rc8.0  Programma in corso
R    yEmission                     ** Emission

LD   yEmission                     ** Emission
ANDN (
LD   Hold_req
AND  PRGRUN_CN0
ANDN %cn0.rc8.1
)
ST   HW_PWM_CFG_FC
ST   INP_laserON                 *** provvisorio
ST   Memo_Emission_ON_da_Funz_M    ** M107.25 Memoria Emission ON da Funzione M

*******************************************************************************
*   Enable data writing
*   M300 or TstP14.14 (from TabLaser)
*   M301 (from shoot)
*******************************************************************************
CAL  RTRIG_EnVal1(CLK=EnValOut1)   ** (TstP14.14) Abilita Attuazione Valori Uscite
CAL  TRIG_EnVal1_G834(CLK=EnValOut1_G834)   ** (TstP14.14) Abilita Attuazione Valori Uscite
CAL  TRIG_EnVal2_G834(CLK=EnValOut2_G834)   ** (TstP14.14) Abilita Attuazione Valori Uscite
CAL  FTRIG_STOP(CLK=PRGSTOP_CN0)

LD   RTRIG_EnVal1.Q
OR   TRIG_EnVal1_G834.Q
OR   TRIG_EnVal2_G834.Q
OR   FTRIG_STOP.Q
AND  PRGRUN_CN0                    ** M0.0 cn0.rc8.0  Programma in corso
ST   appoggio

LD   %cn0.rc9                * Registro funzioni M canale 0
EQ   300
AND  %cn0.rc8.4              * Strobe funzioni M canale 0
OR   appoggio
JMPCN COPYVAL

****************************************
*   TabLsr[]
*   -POWER
*   -DUTY
*   -FREQ
****************************************
LD   xPower                        ** Power
ST   tmpPowerLaserCmd              ** Power temp commanded

LD   xDuty                         ** Duty
ST   tmpDutyLaserCmd

LD   xFreq                         ** Frequency
ST   tmpFreqLaserOut               ** Freq temp

COPYVAL:
****************************************
*   SHOOT
*   -POWER
*   -DUTY
*   -FREQ
****************************************
LD   %cn0.rc9                * Registro funzioni M canale 0
EQ   301
AND  %cn0.rc8.4              * Strobe funzioni M canale 0
JMPCN COPYVAL2

LD   %ShootPower
ST   tmpPowerLaserCmd              ** Power temp commanded

LD   %ShootDuty
ST   tmpDutyLaserCmd

LD   %ShootFreq
ST   tmpFreqLaserOut               ** Freq temp
JMP  COPYVAL3

COPYVAL2:

LD   bevAngleHead1_calc1
ABS
LE   8000
AND (
LD   bevAngleHead1_calc1
ABS
GE   -8000
)
AND  Gest5Ax
ORN  Gest5Ax
AND  L_SOURCE16.9                   * Abilitazione velocità in funzione angolo
ORN  L_SOURCE16.9                   * Abilitazione velocità in funzione angolo
ST   corr_funz_speed

********************************************************************************
********************************************************************************
********************************************************************************
*                               POWER
********************************************************************************
********************************************************************************
********************************************************************************

***************************************
*   Power=func(speed)
***************************************
LD   tmpPowerLaserCmd              ** Power temp commanded
ST   tmpPowerLaserOut              ** Power temp calculated

LD   L_SOURCE16.3                   * Enable POWER management by speed
ANDN (
LD   piercing_run                  ** (LsPlc37) Piercing in run
EQ   1
)
ANDN %ServiceMillePGM.0             * Laser Shoot-on
AND  corr_funz_speed
JMPCN cal_power_speed

LD  PercInterpSpeed
ST  PowerCalc.xPercSpeed           * Speed percentual value (% * 1000)

LD  CurrentLineExecute             ** (LsIso11) Current cutting line parameter to execute
ST  PowerCalc.xCutLineInd          * cut line index (initial value 1 to 10)

LD  1
ST  PowerCalc.xCodTec             * Tecnology 0=duty 1=power 2=frequency

CAL PowerCalc

LD   PowerCalc.yResult             * Result (% * 1000)
DIV  1000
MUL  tmpPowerLaserCmd
DIV  100
ST   tmpPowerLaserOut              ** Power temp calculated

cal_power_speed:

LD   tmpPowerLaserOut
ST   %M65       * TODO (per TEST anche in DRYRUN!)

***************************************
*   Power=func(angle)
*   #CDL
***************************************
LD   PRGRUN_CN0
ANDN PRGSTOP_CN0
AND (
LD   %uvHeads0.uvhCommand1
EQ   4                              * Cutting phase
)
JMPCN no_pow_dataint

LD   tmpPowerLaserOut
ADD (
LD   tmpPowerLaserOut
MULDIV(M=%TsCutDataLinear.CDL_Power, D=100000) * 100 %
)
ST   tmpPowerLaserOut              ** Power temp calculated

no_pow_dataint:

LD   tmpPowerLaserOut
ST   %M66       * TODO (per TEST anche in DRYRUN!)

***************************************
*   Power
*   #INC/DEC MANUALE
***************************************
LD   tmpPowerLaserOut
MUL (
LD   ManSelectorPOW         *(rgGui7)Selettore manuale POTENZA: ultimo valore impostato
SUB  100                    * 100%
)
DIV  100                    * 100 %
ST   ManSelectorPOW_out         *(gPlc30)Selettore manuale POTENZA: ultimo valore impostato (valore di uscita per LsrGest)

***************************************
*   Power linearization
***************************************
LD   LASER_POWER_LINEAR_PAR
JMPCN no_power_an_lin

LD   tmpPowerLaserOut
MUL  1000
ST   PowerLin.xInput

LD   129
ST   PowerLin.xIndex

CAL  PowerLin

LD   PowerLin.yResult            * Result
EQ   2147483647
JMPCN DatoOk

LD   0
ST   tmpPowerLaserOut              ** Power temp calculated
JMP  no_power_an_lin

DatoOk:
LD   PowerLin.yResult            * Result
DIV  1000
ST   tmpPowerLaserOut              ** Power temp calculated

no_power_an_lin:

***************************************

LD   tmpPowerLaserOut
ADD  ManSelectorPOW_out
ST   appoggio_pow

LD   appoggio_pow
GT   LASER_MAX_POWER_PAR
JMPCN NoOutLimits

LD   LASER_MAX_POWER_PAR
ST   appoggio_pow

NoOutLimits:

********************************************************************************
********************************************************************************
********************************************************************************
*                               DUTY
********************************************************************************
********************************************************************************
********************************************************************************

***************************************
*   Duty=func(speed)
***************************************
LD   tmpDutyLaserCmd
ST   tmpDutyLaserOut

LD   L_SOURCE16.2               * Enable DUTY management by speed
ANDN (
LD   piercing_run                  ** (LsPlc37) Piercing in run
EQ   1
)
ANDN %ServiceMillePGM.0             * Laser Shoot-on
AND  corr_funz_speed
JMPCN cal_duty_speed

LD  PercInterpSpeed2
ST  DutyCalc.xPercSpeed          * Speed percentual value

LD  CurrentLineExecute             ** (LsIso11) Current cutting line parameter to execute
ST  DutyCalc.xCutLineInd         * cut line index (initial value 1 to 10)

LD  0
ST  DutyCalc.xCodTec             * Tecnology 0=duty 1=power 2=frequency

CAL DutyCalc

LD  DutyCalc.yResult             * Result
DIV 1000
ST  tmpDutyLaserOut                ** Duty temp

cal_duty_speed:

LD  tmpDutyLaserOut
ST   %M65

***************************************
*   Duty=funz(angle)
*   #CDL
***************************************
LD   PRGRUN_CN0
ANDN PRGSTOP_CN0
AND (
LD   %uvHeads0.uvhCommand1
EQ   4                              * Cutting phase
)
JMPCN no_duty_dataint

LD   tmpDutyLaserOut
ADD (
LD   tmpDutyLaserOut
MULDIV(M=%TsCutDataLinear.CDL_Duty,D=100000) * 100 %
)
ST   tmpDutyLaserOut

no_duty_dataint:
LD  tmpDutyLaserOut
ST   %M66

***************************************
*   DUTY
*   #INC/DEC MANUALE
***************************************
LD   tmpDutyLaserOut
MUL (
LD   ManSelectorDUTY        *(rgGui8)Selettore manuale DUTY: ultimo valore impostato
SUB  100                    * 100%
)
DIV  100                    * 100 %
ST   ManSelectorDUTY_out        *(gPlc30)Selettore manuale DUTY: ultimo valore impostato (valore di uscita per LsrGest)

***************************************
LD   tmpDutyLaserOut               ** Duty temp
ADD  ManSelectorDUTY_out        *(gPlc30)Selettore manuale DUTY: ultimo valore impostato (valore di uscita per LsrGest)
ST   appoggio_duty

LD   appoggio_duty
GT   100
JMPCN no_out_duty

LD   100
ST   appoggio_duty

no_out_duty:

********************************************************************************
********************************************************************************
********************************************************************************
*                               FREQUENCY
********************************************************************************
********************************************************************************
********************************************************************************
LD   L_SOURCE16.4               * Enable FREQUENCY management by speed
ANDN (
LD   piercing_run                  ** (LsPlc37) Piercing in run
EQ   1
)
ANDN %ServiceMillePGM.0             * Laser Shoot-on
JMPCN cal_freq_speed

LD   PercInterpSpeed3
ST   FreqCalc.xPercSpeed           * Speed percentual value

LD   CurrentLineExecute            ** (LsIso11) Current cutting line parameter to execute
ST   FreqCalc.xCutLineInd          * cut line index (initial value 1 to 10)

LD   2
ST   FreqCalc.xCodTec             * Tecnology 0=duty 1=power 2=frequency

CAL  FreqCalc

LD   FreqCalc.yResult             * Result
DIV  100
ST   tmpFreqLaserOut               ** Freq temp

cal_freq_speed:

COPYVAL3:

********************************************************************************
*   Data write >> HW
********************************************************************************
LD   PRGRUN_CN0                    ** M0.0 cn0.rc8.0  Programma in corso
ANDN PRGSTOP_CN0                   ** (cn0.rc8.1)  Programma interrotto CN0
ANDN BCI_RT_DRYRUN                 ** rc64.28 Comando retrace dry run (rapido)
ANDN %PlcOp0.2                     ** DryRun
ANDN LASER_SIM_PAR
ANDN b_TipTouch                    ** (LsPlc47.7) TipTouch Attivo da MainFast
ANDN RETRACERUN                    ** M0.11 Ciclo di retrace in Run
ANDN InibTipTouchAllarm             * Gestione RESTART dopo tip touch
ANDN EnPosiz                       * (LsPlc47.3) Abilitaz. posiz. Asse Z
***ANDN JogCommandTipTouch             * Gestione RESTART dopo tip touch
ANDN Duty0WhenHoldSup                * To avoid shooting laser before M851
JMPC EN_DATA

LD   0
ST   tmpPowerLaserOut              ** Power temp calculated
ST   tmpDutyLaserOut               ** Duty temp
ST   tmpFreqLaserOut               ** Freq temp
ST   appoggio_pow
ST   appoggio_duty

EN_DATA:

*** POWER ***

LD   LASER_POWER_ONBUS_PAR
JMPCN NoOnBus

LD   appoggio_pow
ST   OA_POTENZA_LASER
JMP  ComP

NoOnBus:
LD   appoggio_pow
MUL  LASER_DAC_RES_PAR
DIV  LASER_MAX_POWER_PAR
ST   OA_POTENZA_LASER

ComP:

*** DUTY ***

LD   LASER_USE_PWM_POWER
JMPCN PowerPortNotOnPwm

LD   OA_POTENZA_LASER
ST   HW_PWM_POWER

PowerPortNotOnPwm:

LD   appoggio_duty
MUL  255
DIV  100
AND  16#0fff
ST   HW_PWM_DUTY           ** (QW908)Regolazione Duty Cycle Potenza Laser

*** FREQ. ***

LD   tmpFreqLaserOut               ** Freq temp
ADD  ManSelectorFREQ_out        *(gPlc30)Selettore manuale FREQUENCY: ultimo valore impostato (valore di uscita per LsrGest)
ST   HW_FREQ            ** (QW909)Regolazione Frequenza Potenza Laser

* PWM_RES
LD   255
ST   HW_PWM_RES                    ** (QW910)Impostazione scheda PWM - Reset

****************************************
*   HMI: Data visualization
****************************************
LD   appoggio_pow
ST   %VisPowerOut

LD   appoggio_duty
ST   %VisDutyOut

LD   tmpFreqLaserOut               ** Freq temp
ST   %VisFreqOut

********************************************************************************

********************************************************************************
* *** VAR_IN_OUT WARNING : Latch INP_flyCutModeON to OUT_ before using !     ***
* *** HW ASSISTED FLYCUT : Wait for status register instead !                ***
********************************************************************************

LDN  PRGSTOP_CN0                   ** (cn0.rc8.1)  Programma interrotto CN0
ANDN Pul_Reset                     ** (gPlc0.3)Reset pushbutton
ANDN M_HOLD                        ** (gPlc19.0)Mem. Richiesta Hold
ANDN b_TipTouch                    ** (LsPlc47.7) TipTouch Attivo da MainFast
OR   (
LDN   Touch_enab                   ** C99.8 touch enable
ANDN  Regol_enab                   ** C99.9 regulator enable
AND   %cn0.rc8.0
)
ST   outputEnableON                ** Actually enable output (/pgm interrupted, etc..)

*************************************************
* Protection for fly cut board old version
*************************************************
CAL TOF_Pul_Stop(IN:= Pul_Stop,PT:=500) ** (gPlc0.2)Stop pushbutton

LD   shoot_fly_on                  ** to disable shoot in hold during fly cut old board
AND  OUT_isFlyCutModeON
AND  outputEnableON                ** Actually enable output (/pgm interrupted, etc..)
ANDN TOF_Pul_Stop.Q
JMPCN enable_fly_shot
LD   ALWAYS_ONE                    ** PLCFLAGS.1  Flag sempre stato on
ST   HW_PWM_CFG_FC

LD   ALWAYS_ZERO                   ** PLCFLAGS.0  Flag sempre stato off
ST   shoot_fly_on                  ** to disable shoot in hold during fly cut old board
enable_fly_shot:

LD   OUT_isFlyCutModeON
AND  TOF_Pul_Stop.Q
JMPCN no_output_check
LD   HW_PWM_CFG_FC
S    shoot_fly_on                  ** to disable shoot in hold during fly cut old board
no_output_check:

LD   shoot_fly_on                  ** to disable shoot in hold during fly cut old board
JMPCN force_zero_fly
LD    ALWAYS_ZERO                  ** PLCFLAGS.0  Flag sempre stato off
ST    HW_PWM_CFG_FC
force_zero_fly:

LDN   %cn0.rc8.0
OR    Pul_Reset                    ** (gPlc0.3)Reset pushbutton
JMPCN reset_shoot_fly
LD    ALWAYS_ZERO                  ** PLCFLAGS.0  Flag sempre stato off
ST    shoot_fly_on                 ** to disable shoot in hold during fly cut old board
reset_shoot_fly:

*************************************************
**************************

LD   INP_flyCutModeON   ** application turn flyCut mode ON
ST   OUT_isFlyCutModeON ** application flyCut mode is ON

LD   OUT_isFlyCutModeON ** application flyCut mode is ON
ST   R_TRIG_FC_ON_INIT.CLK

CAL  R_TRIG_FC_ON_INIT

LD   R_TRIG_FC_ON_INIT.Q
ST   flyCutOnInitPulse

LD   OUT_isFlyCutModeON ** application flyCut mode is ON
JMPC flyCutON

LD   PAR_combinedMode   ** use combined PWM and emission
JMPC flyCutOFFcombined

************************************
*** flyCut mode OFF separate PWM ***

LD   0                  ** null bitmap
ST   HW_PWM_CFG         ** Laser I/F board PWM_CFG register      (QW911)

LD   True
ST   HW_PWM_CFG_EN      ** Laser I/F board PWM_CFG register: EN (QW911.0)

LD   INP_laserON        ** application turn laser ON in non-flyCut mode
AND  outputEnableON                ** Actually enable output (/pgm interrupted, etc..)
ST   HW_PWM_CFG_FC      ** Laser I/F board PWM_CFG register: FC (QW911.8)

***                              ***
************************************

JMP  flyCutOFFEND
flyCutOFFcombined:

************************************
*** flyCut mode OFF combined PWM ***

LD   0                  ** null bitmap
ST   HW_PWM_CFG         ** Laser I/F board PWM_CFG register

LD   INP_laserON        ** application turn laser ON in non-flyCut mode
AND  outputEnableON                ** Actually enable output (/pgm interrupted, etc..)
ST   HW_PWM_CFG_EN      ** Laser I/F board PWM_CFG register: EN

***                              ***
************************************

flyCutOFFEND:

JMP  flyCutEND
flyCutON:

LD   PAR_combinedMode   ** use combined PWM and emission
JMPC flyCutONcombined

LD   PAR_TaioEn         ** TAIO flyCut enabled
AND  PAR_TaioAssistEn   ** TAIO Hardware assisted flyCut enabled
JMPC flyCutONseparateHA

************************************
*** flyCut mode ON  separate PWM ***

LD    flyCutOnInitPulse
JMPCN flyCutONseparateEndInit

LD   0                  ** null bitmap
ST   HW_PWM_CFG         ** Laser I/F board PWM_CFG register

LD   True
AND  outputEnableON                ** Actually enable output (/pgm interrupted, etc..)
ST   HW_PWM_CFG_EN      ** Laser I/F board PWM_CFG register: EN

flyCutONseparateEndInit:

***                              ***
************************************

JMP  flyCutONseparateEND
flyCutONseparateHA:

******************************************************
*** flyCut mode ON  separate PWM Hardware Assisted ***

LD   0                  ** null bitmap
ST   HW_PWM_CFG         ** Laser I/F board PWM_CFG register

LD   True
ST   HW_PWM_CFG_EN      ** Laser I/F board PWM_CFG register: EN

LD   True
ST   HW_PWM_CFG_C_EF    ** Laser I/F board PWM_CFG register: C_EF

LD   outputEnableON                ** Actually enable output (/pgm interrupted, etc..)
ST   HW_PWM_CFG_C_OE    ** Laser I/F board PWM_CFG register: C_OE

***                                                ***
******************************************************

flyCutONseparateEND:

JMP  flyCutONEND
flyCutONcombined:

LD   PAR_TaioEn         ** TAIO flyCut enabled
AND  PAR_TaioAssistEn   ** TAIO Hardware assisted flyCut enabled
JMPC flyCutONcombinedHA

************************************
*** flyCut mode ON  combined PWM ***

LD    flyCutOnInitPulse
JMPCN flyCutONcombinedEndInit

LD   0                  ** null bitmap
ST   HW_PWM_CFG         ** Laser I/F board PWM_CFG register

flyCutONcombinedEndInit:

***                              ***
************************************

JMP  flyCutONcombinedEND
flyCutONcombinedHA:

******************************************************
*** flyCut mode ON  combined PWM Hardware Assisted ***

LD   0                  ** null bitmap
ST   HW_PWM_CFG         ** Laser I/F board PWM_CFG register

LD   True
ST   HW_PWM_CFG_C_EF    ** Laser I/F board PWM_CFG register: C_EF
ST   HW_PWM_CFG_C_FR    ** Laser I/F board PWM_CFG register: C_FR

LD   outputEnableON                ** Actually enable output (/pgm interrupted, etc..)
ST   HW_PWM_CFG_C_OE    ** Laser I/F board PWM_CFG register: C_OE

***                                                ***
******************************************************

flyCutONcombinedEND:
flyCutONEND:
flyCutEND:

********************************************************************************
*   GESTIONE LATENZA ON/OFF DIGITAL BEAM PER FLY_CUT
********************************************************************************
LD   %LSRCostK3                    * Valore Costruttore Latenza Attivazione DigitalBeam(Fly_Cut)
ADD  %Cost_User3                   * Valore Personalizz.Utente Latenza Attivazione DigitalBeam(Fly_Cut)
ST   LATENCY_L_TO_H                ** (main_proc.ra77)Latenza Attivazione DigitalBeam FlyCut

LD   %LSRCostK4                    * Valore Costruttore Latenza Disattivazione DigitalBeam(Fly_Cut)
ADD  %Cost_User4                   * Valore Personalizz.Utente Latenza Disattivazione DigitalBeam(Fly_Cut)
ST   LATENCY_H_TO_L                ** (main_proc.ra78)Latenza Disattivazione DigitalBeam FlyCut

LD   EN_T_ALIGNED_SETIO            ** (cg3.23)Opz.CN "Ab.Allineamento SetIo tramite Timer Hardware"
JMPC AZZREAVAL
LD   0
ST   LATENCY_L_TO_H                ** (main_proc.ra77)Latenza Attivazione DigitalBeam FlyCut
ST   LATENCY_H_TO_L                ** (main_proc.ra78)Latenza Disattivazione DigitalBeam FlyCut

AZZREAVAL:
**************************************************************************************************************
**************************************************************************************************************
* Latency for raster print

LD   RasterLatency
ST   %ax21.ra119
**************************************************************************************************************
END_FUNCTION_BLOCK

*******************************************************************************
*   SHOOT management
*******************************************************************************
FUNCTION_BLOCK LASER_SHOOT

VAR_INPUT
xId:        DWORD;          * 0,1
END_VAR

VAR_OUTPUT
yShootOn:   BOOL;
END_VAR

VAR
RTRIG_SHOOT_ON:     R_TRIG;
RTRIG_SHOOT_OFF:    R_TRIG;
FT_PRGRUN:          F_TRIG;
RTRIG_REM_SHOT:     R_TRIG;
CTU_PULS:           CTU;
RTRIG_SHUTTER:      R_TRIG;
FTRIG_SHUTTER:      F_TRIG;
SHUTTER:            BOOL;
appoggio:           BOOL;
END_VAR
*******************************************************************************

***PATH %LsrGest[xId]

CAL  FT_PRGRUN(CLK=PRGRUN_CN0)     ** M0.0 cn0.rc8.0  Programma in corso
CAL  RTRIG_SHOOT_ON(CLK=%lButton0.0)
CAL  RTRIG_SHOOT_OFF(CLK=%lButton0.1)

LD   RemContrShoot
ANDN Rem_Combination
OR   ButtGuiShootLsr
ST   appoggio
CAL  RTRIG_REM_SHOT(CLK:=appoggio)        * Xhc_Puls.17 Laser shut

CAL  CTU_PULS(CU:=RTRIG_REM_SHOT.Q,R=CTU_PULS.Q,PV=2)

LD   CTU_PULS.CV
EQ   1
ST   SHUTTER

CAL  RTRIG_SHUTTER(CLK:=SHUTTER)
CAL  FTRIG_SHUTTER(CLK:=SHUTTER)

LD   RTRIG_SHOOT_ON.Q
*OR   RTRIG_SHUTTER.Q
OR   RTRIG_REM_SHOT.Q
S    %ServiceMillePGM.0

LD   M30_CN0                       ** M0.13 M30:EndProgram CN0
OR   MACC_ALARM                    ** (gPlc0.10)Macchina in allarme
OR   Pul_Reset                     ** (gPlc0.3)Reset pushbutton
OR   FT_PRGRUN.Q
OR   RTRIG_SHOOT_OFF.Q
*OR   FTRIG_SHUTTER.Q
OR   ON_ONE_SCAN                   ** PLCFLAGS.8  Flag on alla prima scansione PLC
R    %ServiceMillePGM.0

LD   %ServiceMillePGM.0
ST   yShootOn

END_FUNCTION_BLOCK
